END_VAR
TEST('TimeoutIncludesEntryAndSatisfiedConditions');
sm.ResetAll(); sm.ForceState(state := TcForge.E_SM_State.RUNNING); sm.SetCurrentStep(nStep := 3000); sm.SetTimerSeconds(seconds := 1.0);
step_TimeoutIncludesEntryAndSatisfiedConditions(sm := sm, nStep := 3000, nNextStep := 3002, nTimeout := 1, nRequired := 0);
AssertFalse(Condition := step_TimeoutIncludesEntryAndSatisfiedConditions.Entry OR step_TimeoutIncludesEntryAndSatisfiedConditions.Execute OR step_TimeoutIncludesEntryAndSatisfiedConditions.Exiting, Message := 'Timeout must suppress all lifecycle outputs even with no missing conditions');
AssertEquals_DINT(Expected := TcForge.E_SM_Fault.StepTimeout, Actual := sm.GetFaultCode(), Message := 'Timeout at the configured boundary');
TEST_FINISHED();
END_METHOD

METHOD StopTimeoutEscalatesToAbort
VAR

END_VAR
TEST('StopTimeoutEscalatesToAbort');
sm.ResetAll(); sm.ForceState(state := TcForge.E_SM_State.STOPPING); sm.SetCurrentStep(nStep := 2000); sm.ForceNextStep(nStep := 2000); sm.SetTimerSeconds(seconds := 2.0);
step_StopTimeoutEscalatesToAbort(sm := sm, nStep := 2000, nNextStep := 0, nTimeout := 1);
sm();
AssertEquals_DINT(Expected := TcForge.E_SM_State.ABORTING, Actual := sm.Status.State, Message := 'Failed Stop must escalate');
AssertEquals_DINT(Expected := 5000, Actual := sm.Status.Step.Current, Message := 'Abort entry step selected immediately');
AssertTrue(Condition := sm.IsFaulted(), Message := 'Escalation must preserve failure diagnostics');
TEST_FINISHED();
END_METHOD

METHOD StopUserFaultEscalatesToAbort
VAR

END_VAR
TEST('StopUserFaultEscalatesToAbort');
sm.ResetAll(); sm.ForceState(state := TcForge.E_SM_State.STOPPING); sm.SetCurrentStep(nStep := 2000); sm.ForceNextStep(nStep := 2000);
step_StopUserFaultEscalatesToAbort(sm := sm, nStep := 2000, nNextStep := 0, nTimeout := 0);
step_StopUserFaultEscalatesToAbort.RaiseFault(code := 101, reason := 'Stop feedback failed'); sm();
AssertEquals_DINT(Expected := TcForge.E_SM_State.ABORTING, Actual := sm.Status.State, Message := 'Custom shutdown fault must escalate independently of diagnostic code');
TEST_FINISHED();
END_METHOD

METHOD AbortTimeoutRequiresConfirmedShutdown
VAR
rsp : TcForge.E_RpcMethodResponse;
END_VAR
TEST('AbortTimeoutRequiresConfirmedShutdown');
sm.ResetAll(); sm.ForceState(state := TcForge.E_SM_State.ABORTING); sm.SetCurrentStep(nStep := 5000); sm.ForceNextStep(nStep := 5000); sm.SetTimerSeconds(seconds := 2.0);
step_AbortTimeoutRequiresConfirmedShutdown(sm := sm, nStep := 5000, nNextStep := 0, nTimeout := 1); sm();
AssertEquals_DINT(Expected := TcForge.E_SM_State.STOPPED, Actual := sm.Status.State, Message := 'Failed Abort must leave a defined terminal state');
AssertTrue(Condition := sm.Status.ShutdownFailed AND sm.IsFaulted(), Message := 'Terminal state must not masquerade as confirmed shutdown');
rsp := sm.Reset();
AssertEquals_DINT(Expected := TcForge.E_RpcMethodResponse.REJECTED_INTERLOCKED, Actual := rsp, Message := 'Reset requires application shutdown confirmation');
sm.inpShutdownConfirmed := TRUE; rsp := sm.Reset();
AssertEquals_DINT(Expected := TcForge.E_RpcMethodResponse.ACCEPTED, Actual := rsp, Message := 'Confirmed healthy terminal shutdown permits Reset');
AssertFalse(Condition := sm.Status.ShutdownFailed OR sm.IsFaulted(), Message := 'Reset clears the latched shutdown diagnostic');
TEST_FINISHED();
END_METHOD

METHOD CustomStepFaultCanRetry
VAR
rsp : TcForge.E_RpcMethodResponse;
END_VAR
TEST('CustomStepFaultCanRetry');
sm.ResetAll(); sm.ForceState(state := TcForge.E_SM_State.RUNNING); sm.SetCurrentStep(nStep := 3000); sm.ForceNextStep(nStep := 3000);
step_CustomStepFaultCanRetry(sm := sm, nStep := 3000, nNextStep := 3002, nTimeout := 0); step_CustomStepFaultCanRetry.RaiseFault(code := 101, reason := 'Application fault'); sm();
rsp := sm.Retry(); AssertEquals_DINT(Expected := TcForge.E_RpcMethodResponse.ACCEPTED, Actual := rsp, Message := 'Recorded custom step faults must support explicit retry');
sm(); sm(); AssertEquals_DINT(Expected := 3000, Actual := sm.Status.Step.Current, Message := 'Retry returns to failed even step');
TEST_FINISHED();
END_METHOD

METHOD MissingActiveStepFaults
VAR

END_VAR
TEST('MissingActiveStepFaults');
missing(); missing.Home(); missing(); missing();
AssertEquals_DINT(Expected := TcForge.E_SM_Fault.MissingStepImplementation, Actual := missing.GetFaultCode(), Message := 'Uncalled active step cannot silently stall');
AssertEquals_DINT(Expected := 1000, Actual := missing.Status.FailedStep, Message := 'Identify the missing implementation');
TEST_FINISHED();
END_METHOD

METHOD DuplicateActiveStepFaults
VAR

END_VAR
TEST('DuplicateActiveStepFaults');
duplicate(); duplicate.Home(); duplicate();
duplicateA(sm := duplicate, nStep := 1000, nNextStep := 0, nTimeout := 0);
duplicateB(sm := duplicate, nStep := 1000, nNextStep := 0, nTimeout := 0);
duplicate();
AssertEquals_DINT(Expected := TcForge.E_SM_Fault.DuplicateStepImplementation, Actual := duplicate.GetFaultCode(), Message := 'Two implementations of the active step must fault');
TEST_FINISHED();
END_METHOD

METHOD MissingDestinationImplementationFaults
VAR
i : INT;
END_VAR
TEST('MissingDestinationImplementationFaults');
missingTarget(); missingTarget.Home(); missingTarget();
FOR i := 1 TO 5 DO
    targetStep(sm := missingTarget, nStep := 1000, nNextStep := 1002, nTimeout := 0);
    missingTarget();
END_FOR;
AssertEquals_DINT(Expected := TcForge.E_SM_Fault.MissingStepImplementation, Actual := missingTarget.GetFaultCode(), Message := 'Valid but unimplemented destination must fault');
AssertEquals_DINT(Expected := 1002, Actual := missingTarget.Status.FailedStep, Message := 'Report destination without implementation');
TEST_FINISHED();
END_METHOD

METHOD MissingAbortImplementationFailsShutdown
VAR

END_VAR
TEST('MissingAbortImplementationFailsShutdown');
missingAbort(); missingAbort.Home(); missingAbort(); missingAbort.Abort(); missingAbort(); missingAbort();
AssertEquals_DINT(Expected := TcForge.E_SM_State.STOPPED, Actual := missingAbort.Status.State, Message := 'Missing Abort cannot leave a stuck state');
AssertTrue(Condition := missingAbort.Status.ShutdownFailed, Message := 'Missing Abort requires confirmed recovery');
TEST_FINISHED();
END_METHOD

METHOD StepZeroNeverExecutes
VAR

END_VAR
TEST('StepZeroNeverExecutes');
zero(); zeroStep(sm := zero, nStep := 0, nNextStep := 0, nTimeout := 0);
AssertFalse(Condition := zeroStep.Entry OR zeroStep.Execute OR zeroStep.Exiting, Message := 'Idle step zero is not executable work');
TEST_FINISHED();
END_METHOD

METHOD TimeoutAboveTimerRangeRejected
VAR

END_VAR
TEST('TimeoutAboveTimerRangeRejected');
sm.ResetAll(); sm.ForceState(state := TcForge.E_SM_State.RUNNING); sm.SetCurrentStep(nStep := 3000);
extraTimeout(sm := sm, nStep := 3000, nNextStep := 0, nTimeout := 356401);
AssertFalse(Condition := extraTimeout.Entry, Message := 'Unsupported timeout cannot silently wait forever');
AssertEquals_DINT(Expected := TcForge.E_SM_Fault.InvalidStepConfiguration, Actual := sm.GetFaultCode(), Message := 'Timeout above timer range is invalid');
TEST_FINISHED();
END_METHOD

METHOD ZeroFaultCodeStillInhibits
VAR

END_VAR
TEST('ZeroFaultCodeStillInhibits');
sm.ResetAll(); sm.ForceState(state := TcForge.E_SM_State.RUNNING); sm.SetCurrentStep(nStep := 3000);
extraZero(sm := sm, nStep := 3000, nNextStep := 0, nTimeout := 0); extraZero.RaiseFault(code := 0, reason := 'Invalid application code');
AssertTrue(Condition := sm.IsFaulted(), Message := 'Zero cannot hide a requested fault');
AssertFalse(Condition := extraZero.Entry OR extraZero.Execute OR extraZero.Exiting, Message := 'Fault immediately removes lifecycle outputs');
AssertEquals_DINT(Expected := TcForge.E_SM_Fault.StepUserFault, Actual := sm.GetFaultCode(), Message := 'Normalize invalid code');
TEST_FINISHED();
END_METHOD

METHOD NegativeFaultCodeStillInhibits
VAR

END_VAR
TEST('NegativeFaultCodeStillInhibits');
sm.ResetAll(); sm.ForceState(state := TcForge.E_SM_State.RUNNING); sm.SetCurrentStep(nStep := 3000);
extraNegative(sm := sm, nStep := 3000, nNextStep := 0, nTimeout := 0); extraNegative.RaiseFault(code := -1, reason := 'Invalid application code');
AssertTrue(Condition := sm.IsFaulted(), Message := 'Negative code cannot hide a requested fault');
AssertEquals_DINT(Expected := TcForge.E_SM_Fault.StepUserFault, Actual := sm.GetFaultCode(), Message := 'Normalize invalid code');
TEST_FINISHED();
END_METHOD

METHOD InvalidResetPreservesShutdownLatch
VAR
raw : DINT := 99;
requester : POINTER TO TcForge.E_Requester;
rsp : TcForge.E_RpcMethodResponse;
END_VAR
TEST('InvalidResetPreservesShutdownLatch');
sm.ResetAll(); sm.ForceState(state := TcForge.E_SM_State.ABORTING); sm.SetCurrentStep(nStep := 5000); sm.ForceNextStep(nStep := 5000);
extraReset(sm := sm, nStep := 5000, nNextStep := 0, nTimeout := 0); extraReset.RaiseFault(code := 101, reason := 'Abort failed'); sm();
sm.inpShutdownConfirmed := TRUE;
requester := ADR(raw); rsp := sm.Reset(eRequester := requester^);
AssertEquals_DINT(Expected := TcForge.E_RpcMethodResponse.REJECTED_INVALID_PARAMETER, Actual := rsp, Message := 'Invalid command identity rejected');
AssertTrue(Condition := sm.Status.ShutdownFailed, Message := 'Rejected reset preserves shutdown latch');
AssertEquals_DINT(Expected := 5000, Actual := sm.Status.FailedStep, Message := 'Rejected reset preserves failed step');
TEST_FINISHED();
END_METHOD

END_FUNCTION_BLOCK

// ---- Testing/Tests/FB_Foundation_Test.TcPOU
FUNCTION_BLOCK FB_Foundation_Test EXTENDS TcUnit.FB_TestSuite
VAR
    _done : BOOL;
    RecordedFaultBlocksStart_sm : FB_StateMachine_Probe;
    RetryRecoversOddStep_sm : FB_StateMachine_Probe;
    StopHandlesPausedAndHoming_sm : FB_StateMachine_Probe;
    AbortCannotBeOverwritten_sm : FB_StateMachine_Probe;
    StopCancelsQueuedHome_sm : FB_StateMachine_Probe;
    PendingHomeRechecksPermissive_sm : FB_StateMachine_Probe;
    MissingRequiredPermissiveInhibits_fb : TcForge.FB_Permissives;
    MissingRequiredInterlockLatches_fb : TcForge.FB_Interlock;
    DigitalQualityRecoveryNeedsCommand_fb : TcForge.FB_DigitalOutput;
    ForceSafeBypassesInvertAndDelay_fb : TcForge.FB_DigitalOutput;
    OperatorCannotClaimProgram_fb : TcForge.FB_DigitalOutput;
    AnalogLiveConfigFaultInhibits_fb : TcForge.FB_AnalogOutput;
    AnalogQualityRecoveryNeedsCommand_fb : TcForge.FB_AnalogOutput;
    ActuatorTripDropsOutputSameScan_fb : TcForge.FB_TwoPosActuator;
    ActuatorAbortDoesNotReenergizeHold_fb : TcForge.FB_TwoPosActuator;
    ExternalInputUsesPublicBoundary_fb : TcForge.FB_DigitalInput;
    ResetDoesNotStopRunningMachine_sm : FB_StateMachine_Probe;
    PublicSequenceLifecycle_sm : TcForge.FB_StateMachine;
    PublicSequenceLifecycle_homeStep : TcForge.FB_Step;
    PublicSequenceLifecycle_stopStep : TcForge.FB_Step;
    RateAlarmSeedsAndDetectsChange_fb : TcForge.FB_AlarmRateOfChange;
    StartupDoesNotRestoreWithoutOptIn_fb : FB_OutputRestart_Probe;
    StartupRestoreRequiresGoodQuality_fb : FB_OutputRestart_Probe;
    StartupRestoreRequiresGoodQuality_restored : FB_OutputRestart_Probe;
    SubmoduleFaultDoesNotPreventAbortCompletion_sm : FB_StateMachine_Probe;
    ActuatorAbortDominatesSameScan_fb : TcForge.FB_TwoPosActuator;
END_VAR

IF _done THEN RETURN; END_IF;
RecordedFaultBlocksStart();
RetryRecoversOddStep();
StopHandlesPausedAndHoming();
AbortCannotBeOverwritten();
StopCancelsQueuedHome();
PendingHomeRechecksPermissive();
MissingRequiredPermissiveInhibits();
MissingRequiredInterlockLatches();
DigitalQualityRecoveryNeedsCommand();
ForceSafeBypassesInvertAndDelay();
OperatorCannotClaimProgram();
AnalogLiveConfigFaultInhibits();
AnalogQualityRecoveryNeedsCommand();
ActuatorTripDropsOutputSameScan();
ActuatorAbortDoesNotReenergizeHold();
ExternalInputUsesPublicBoundary();
ResetDoesNotStopRunningMachine();
PublicSequenceLifecycle();
RateAlarmSeedsAndDetectsChange();
StartupDoesNotRestoreWithoutOptIn();
StartupRestoreRequiresGoodQuality();
SubmoduleFaultDoesNotPreventAbortCompletion();
ActuatorAbortDominatesSameScan();
_done := TRUE;

METHOD RecordedFaultBlocksStart
VAR
rsp : TcForge.E_RpcMethodResponse;
END_VAR
TEST('RecordedFaultBlocksStart');
RecordedFaultBlocksStart_sm.ResetAll(); RecordedFaultBlocksStart_sm.ForceState(state := TcForge.E_SM_State.READY); RecordedFaultBlocksStart_sm();
RecordedFaultBlocksStart_sm.inpSubmoduleFaulted := TRUE; RecordedFaultBlocksStart_sm();
rsp := RecordedFaultBlocksStart_sm.Start();
AssertEquals_DINT(Expected := TcForge.E_RpcMethodResponse.REJECTED_FAULTED, Actual := rsp, Message := 'Base fault must block Start even on an even step');
TEST_FINISHED();
END_METHOD

METHOD RetryRecoversOddStep
VAR
rsp : TcForge.E_RpcMethodResponse;
END_VAR
TEST('RetryRecoversOddStep');
RetryRecoversOddStep_sm.ResetAll(); RetryRecoversOddStep_sm.ForceState(state := TcForge.E_SM_State.RUNNING);
RetryRecoversOddStep_sm.SetCurrentStep(nStep := 3001); RetryRecoversOddStep_sm.ForceNextStep(nStep := 3001); RetryRecoversOddStep_sm();
rsp := RetryRecoversOddStep_sm.Retry();
AssertEquals_DINT(Expected := TcForge.E_RpcMethodResponse.ACCEPTED, Actual := rsp, Message := 'Retry must accept recovery step');
RetryRecoversOddStep_sm(); RetryRecoversOddStep_sm();
AssertEquals_DINT(Expected := 3000, Actual := RetryRecoversOddStep_sm.Status.Step.Current, Message := 'Retry re-enters previous even step');
AssertFalse(Condition := RetryRecoversOddStep_sm.IsFaulted(), Message := 'Recovered step fault must clear');
TEST_FINISHED();
END_METHOD

METHOD StopHandlesPausedAndHoming
VAR
i : INT;
rsp : TcForge.E_RpcMethodResponse;
END_VAR
TEST('StopHandlesPausedAndHoming');
FOR i := 0 TO 1 DO
StopHandlesPausedAndHoming_sm.ResetAll();
IF i = 0 THEN StopHandlesPausedAndHoming_sm.ForceState(state := TcForge.E_SM_State.PAUSED); ELSE StopHandlesPausedAndHoming_sm.ForceState(state := TcForge.E_SM_State.HOMING); END_IF;
rsp := StopHandlesPausedAndHoming_sm.Stop(); StopHandlesPausedAndHoming_sm();
AssertEquals_DINT(Expected := TcForge.E_RpcMethodResponse.ACCEPTED, Actual := rsp, Message := 'Stop is accepted');
AssertEquals_DINT(Expected := TcForge.E_SM_State.STOPPING, Actual := StopHandlesPausedAndHoming_sm.Status.State, Message := 'Accepted Stop starts stopping sequence');
END_FOR;
TEST_FINISHED();
END_METHOD

METHOD AbortCannotBeOverwritten
VAR
rsp : TcForge.E_RpcMethodResponse;
END_VAR
TEST('AbortCannotBeOverwritten');
AbortCannotBeOverwritten_sm.ResetAll(); AbortCannotBeOverwritten_sm.ForceState(state := TcForge.E_SM_State.RUNNING);
AbortCannotBeOverwritten_sm.Abort(); rsp := AbortCannotBeOverwritten_sm.Pause(); AbortCannotBeOverwritten_sm.Stop(); AbortCannotBeOverwritten_sm();
AssertEquals_DINT(Expected := TcForge.E_RpcMethodResponse.REJECTED_WRONG_STATE, Actual := rsp, Message := 'Pause cannot replace Abort');
AssertEquals_DINT(Expected := TcForge.E_SM_State.ABORTING, Actual := AbortCannotBeOverwritten_sm.Status.State, Message := 'Abort has priority');
TEST_FINISHED();
END_METHOD

METHOD StopCancelsQueuedHome
VAR
END_VAR
TEST('StopCancelsQueuedHome');
StopCancelsQueuedHome_sm.ResetAll(); StopCancelsQueuedHome_sm(); StopCancelsQueuedHome_sm.Home(); StopCancelsQueuedHome_sm.Stop(); StopCancelsQueuedHome_sm(); StopCancelsQueuedHome_sm();
AssertEquals_DINT(Expected := TcForge.E_SM_State.STOPPED, Actual := StopCancelsQueuedHome_sm.Status.State, Message := 'Queued home must not survive Stop');
TEST_FINISHED();
END_METHOD

METHOD PendingHomeRechecksPermissive
VAR
END_VAR
TEST('PendingHomeRechecksPermissive');
PendingHomeRechecksPermissive_sm.ResetAll(); PendingHomeRechecksPermissive_sm(); PendingHomeRechecksPermissive_sm.Home(); PendingHomeRechecksPermissive_sm.MapHomeCondition(bitIndex := 0, bGood := FALSE); PendingHomeRechecksPermissive_sm();
AssertEquals_DINT(Expected := TcForge.E_SM_State.STOPPED, Actual := PendingHomeRechecksPermissive_sm.Status.State, Message := 'Current bad permission cancels pending Home');
PendingHomeRechecksPermissive_sm.MapHomeCondition(bitIndex := 0, bGood := TRUE); PendingHomeRechecksPermissive_sm();
AssertEquals_DINT(Expected := TcForge.E_SM_State.STOPPED, Actual := PendingHomeRechecksPermissive_sm.Status.State, Message := 'Cancelled request must not restart later');
TEST_FINISHED();
END_METHOD

METHOD MissingRequiredPermissiveInhibits
VAR
i : INT;
END_VAR
TEST('MissingRequiredPermissiveInhibits');
MissingRequiredPermissiveInhibits_fb.cfg.nRequired := 1; MissingRequiredPermissiveInhibits_fb();
AssertFalse(Condition := MissingRequiredPermissiveInhibits_fb.sts.bOK, Message := 'Never-mapped required condition must inhibit');
MissingRequiredPermissiveInhibits_fb.MapInput(bitIndex := 0, inputValue := TRUE); MissingRequiredPermissiveInhibits_fb();
AssertTrue(Condition := MissingRequiredPermissiveInhibits_fb.sts.bOK, Message := 'Fresh required condition is good');
FOR i := 1 TO 12 DO MissingRequiredPermissiveInhibits_fb(); END_FOR;
AssertFalse(Condition := MissingRequiredPermissiveInhibits_fb.sts.bOK, Message := 'Stale required condition must inhibit');
AssertEquals_ULINT(Expected := 1, Actual := MissingRequiredPermissiveInhibits_fb.sts.nMissing, Message := 'Missing mask identifies condition');
TEST_FINISHED();
END_METHOD

METHOD MissingRequiredInterlockLatches
VAR
i : INT;
END_VAR
TEST('MissingRequiredInterlockLatches');
MissingRequiredInterlockLatches_fb.cfg.nRequired := 1; MissingRequiredInterlockLatches_fb.MapInput(bitIndex := 0, inputValue := TRUE); MissingRequiredInterlockLatches_fb();
FOR i := 1 TO 12 DO MissingRequiredInterlockLatches_fb(); END_FOR;
MissingRequiredInterlockLatches_fb.MapInput(bitIndex := 0, inputValue := TRUE); MissingRequiredInterlockLatches_fb();
AssertFalse(Condition := MissingRequiredInterlockLatches_fb.sts.bOK, Message := 'Recovered missing interlock requires Reset');
MissingRequiredInterlockLatches_fb.Reset(); MissingRequiredInterlockLatches_fb.MapInput(bitIndex := 0, inputValue := TRUE); MissingRequiredInterlockLatches_fb();
AssertTrue(Condition := MissingRequiredInterlockLatches_fb.sts.bOK, Message := 'Reset after fresh data releases missing latch');
TEST_FINISHED();
END_METHOD

METHOD DigitalQualityRecoveryNeedsCommand
VAR
END_VAR
TEST('DigitalQualityRecoveryNeedsCommand');
DigitalQualityRecoveryNeedsCommand_fb.SetOn(); DigitalQualityRecoveryNeedsCommand_fb(); AssertTrue(Condition := DigitalQualityRecoveryNeedsCommand_fb.sts.value, Message := 'Output starts on command');
DigitalQualityRecoveryNeedsCommand_fb(inpQuality := TcForge.E_IO_Quality.BAD);
AssertFalse(Condition := DigitalQualityRecoveryNeedsCommand_fb.sts.value, Message := 'Default bad-quality policy applies safe level');
DigitalQualityRecoveryNeedsCommand_fb(inpQuality := TcForge.E_IO_Quality.GOOD);
AssertFalse(Condition := DigitalQualityRecoveryNeedsCommand_fb.sts.value, Message := 'Quality recovery alone must not energize');
DigitalQualityRecoveryNeedsCommand_fb.SetOn(); DigitalQualityRecoveryNeedsCommand_fb(); AssertTrue(Condition := DigitalQualityRecoveryNeedsCommand_fb.sts.value, Message := 'Fresh command resumes output');
TEST_FINISHED();
END_METHOD

METHOD ForceSafeBypassesInvertAndDelay
VAR
rsp : TcForge.E_RpcMethodResponse;
END_VAR
TEST('ForceSafeBypassesInvertAndDelay');
ForceSafeBypassesInvertAndDelay_fb.cfg.invert := TRUE; ForceSafeBypassesInvertAndDelay_fb.cfg.debounceOff := T#10S;
ForceSafeBypassesInvertAndDelay_fb.SetOff(); ForceSafeBypassesInvertAndDelay_fb(); ForceSafeBypassesInvertAndDelay_fb.ForceSafe(); rsp := ForceSafeBypassesInvertAndDelay_fb.SetOn(); ForceSafeBypassesInvertAndDelay_fb();
AssertEquals_DINT(Expected := TcForge.E_RpcMethodResponse.REJECTED_INTERLOCKED, Actual := rsp, Message := 'ForceSafe wins within scan');
AssertFalse(Condition := ForceSafeBypassesInvertAndDelay_fb.sts.value, Message := 'ForceSafe writes electrical safe level without invert/delay');
TEST_FINISHED();
END_METHOD

METHOD OperatorCannotClaimProgram
VAR
rsp : TcForge.E_RpcMethodResponse;
END_VAR
TEST('OperatorCannotClaimProgram');
OperatorCannotClaimProgram_fb();
OperatorCannotClaimProgram_fb.LockSource(bLock := TRUE); rsp := OperatorCannotClaimProgram_fb.OperatorSetOn(requestId := 1);
AssertEquals_DINT(Expected := TcForge.E_RpcMethodResponse.QUEUED, Actual := rsp, Message := 'Admission is not execution');
OperatorCannotClaimProgram_fb();
rsp := OperatorCannotClaimProgram_fb.OperatorCommandResult(requestId := 1);
AssertEquals_DINT(Expected := TcForge.E_RpcMethodResponse.REJECTED_SOURCE_NOT_ALLOWED, Actual := rsp, Message := 'Operator wrapper always uses OPERATOR identity');
TEST_FINISHED();
END_METHOD

METHOD AnalogLiveConfigFaultInhibits
VAR
END_VAR
TEST('AnalogLiveConfigFaultInhibits');
AnalogLiveConfigFaultInhibits_fb.SetValue(rValue := 50.0); AnalogLiveConfigFaultInhibits_fb(); AnalogLiveConfigFaultInhibits_fb.cfg.euMax := AnalogLiveConfigFaultInhibits_fb.cfg.euMin; AnalogLiveConfigFaultInhibits_fb();
AssertTrue(Condition := AnalogLiveConfigFaultInhibits_fb.IsFaulted(), Message := 'Live invalid range must fault');
AssertTrue(Condition := AnalogLiveConfigFaultInhibits_fb.sts.outputInhibited, Message := 'Invalid config inhibits output same scan');
AssertTrue(Condition := AnalogLiveConfigFaultInhibits_fb.sts.rawReal = 0.0, Message := 'Fallback is raw safe value');
TEST_FINISHED();
END_METHOD

METHOD AnalogQualityRecoveryNeedsCommand
VAR
END_VAR
TEST('AnalogQualityRecoveryNeedsCommand');
AnalogQualityRecoveryNeedsCommand_fb.SetValue(rValue := 50.0); AnalogQualityRecoveryNeedsCommand_fb(); AnalogQualityRecoveryNeedsCommand_fb(inpQuality := TcForge.E_IO_Quality.UNKNOWN); AnalogQualityRecoveryNeedsCommand_fb(inpQuality := TcForge.E_IO_Quality.GOOD);
AssertTrue(Condition := AnalogQualityRecoveryNeedsCommand_fb.sts.outputInhibited, Message := 'Unknown quality disarms until fresh command');
AnalogQualityRecoveryNeedsCommand_fb.SetValue(rValue := 25.0); AnalogQualityRecoveryNeedsCommand_fb();
AssertFalse(Condition := AnalogQualityRecoveryNeedsCommand_fb.sts.outputInhibited, Message := 'Fresh command re-arms');
TEST_FINISHED();
END_METHOD

METHOD ActuatorTripDropsOutputSameScan
VAR
END_VAR
TEST('ActuatorTripDropsOutputSameScan');
ActuatorTripDropsOutputSameScan_fb(inAdvanced := FALSE, inRetracted := TRUE);
ActuatorTripDropsOutputSameScan_fb.Advance(); ActuatorTripDropsOutputSameScan_fb(); AssertTrue(Condition := ActuatorTripDropsOutputSameScan_fb.outAdvance, Message := 'Motion output energized');
ActuatorTripDropsOutputSameScan_fb(inAdvanced := TRUE, inRetracted := TRUE);
AssertTrue(Condition := ActuatorTripDropsOutputSameScan_fb.IsFaulted(), Message := 'Contradictory feedback faults');
AssertFalse(Condition := ActuatorTripDropsOutputSameScan_fb.outAdvance OR ActuatorTripDropsOutputSameScan_fb.outRetract, Message := 'Fault removes both outputs same scan');
TEST_FINISHED();
END_METHOD

METHOD ActuatorAbortDoesNotReenergizeHold
VAR
END_VAR
TEST('ActuatorAbortDoesNotReenergizeHold');
ActuatorAbortDoesNotReenergizeHold_fb.cfg.holdAtRetracted := TRUE; ActuatorAbortDoesNotReenergizeHold_fb(inRetracted := TRUE);
ActuatorAbortDoesNotReenergizeHold_fb.Abort(); ActuatorAbortDoesNotReenergizeHold_fb(); ActuatorAbortDoesNotReenergizeHold_fb();
AssertFalse(Condition := ActuatorAbortDoesNotReenergizeHold_fb.outRetract, Message := 'Abort must not automatically energize hold coil later');
TEST_FINISHED();
END_METHOD

METHOD ExternalInputUsesPublicBoundary
VAR
END_VAR
TEST('ExternalInputUsesPublicBoundary');
ExternalInputUsesPublicBoundary_fb(inSignal := TRUE);
AssertTrue(Condition := ExternalInputUsesPublicBoundary_fb.sts.value, Message := 'Digital external input path works without probe');
TEST_FINISHED();
END_METHOD

METHOD ResetDoesNotStopRunningMachine
VAR
rsp : TcForge.E_RpcMethodResponse;
END_VAR
TEST('ResetDoesNotStopRunningMachine');
ResetDoesNotStopRunningMachine_sm.ResetAll(); ResetDoesNotStopRunningMachine_sm.ForceState(state := TcForge.E_SM_State.RUNNING); rsp := ResetDoesNotStopRunningMachine_sm.Reset();
AssertEquals_DINT(Expected := TcForge.E_RpcMethodResponse.REJECTED_WRONG_STATE, Actual := rsp, Message := 'Reset requires stopped state');
TEST_FINISHED();
END_METHOD

METHOD PublicSequenceLifecycle
VAR
i : INT;
END_VAR
TEST('PublicSequenceLifecycle');
PublicSequenceLifecycle_sm(); PublicSequenceLifecycle_sm.Home(); PublicSequenceLifecycle_sm();
AssertEquals_DINT(Expected := 1000, Actual := PublicSequenceLifecycle_sm.Status.Step.Current, Message := 'Home enters first step');
FOR i := 1 TO 5 DO
    PublicSequenceLifecycle_homeStep(sm := PublicSequenceLifecycle_sm, nStep := 1000, nNextStep := 0, nTimeout := 0, sName := 'Home'); PublicSequenceLifecycle_sm();
END_FOR;
AssertEquals_DINT(Expected := TcForge.E_SM_State.READY, Actual := PublicSequenceLifecycle_sm.Status.State, Message := 'Home completion enters ready');
PublicSequenceLifecycle_sm.Start(); PublicSequenceLifecycle_sm(); PublicSequenceLifecycle_sm.Stop(); PublicSequenceLifecycle_sm();
FOR i := 1 TO 5 DO
    PublicSequenceLifecycle_stopStep(sm := PublicSequenceLifecycle_sm, nStep := 2000, nNextStep := 0, nTimeout := 0, sName := 'Stop'); PublicSequenceLifecycle_sm();
END_FOR;
AssertEquals_DINT(Expected := TcForge.E_SM_State.STOPPED, Actual := PublicSequenceLifecycle_sm.Status.State, Message := 'Stop sequence completes through public API');
PublicSequenceLifecycle_sm(); AssertEquals_DINT(Expected := TcForge.E_SM_State.STOPPED, Actual := PublicSequenceLifecycle_sm.Status.State, Message := 'No stale commands replay');
TEST_FINISHED();
END_METHOD

METHOD RateAlarmSeedsAndDetectsChange
VAR
END_VAR
TEST('RateAlarmSeedsAndDetectsChange');
RateAlarmSeedsAndDetectsChange_fb.cfg.common.bEnable := TRUE; RateAlarmSeedsAndDetectsChange_fb.cfg.fRateLimit := 1.0;
RateAlarmSeedsAndDetectsChange_fb(inpPv := 100.0); AssertTrue(Condition := RateAlarmSeedsAndDetectsChange_fb.outRateOfChange = 0.0, Message := 'First scan seeds rate');
RateAlarmSeedsAndDetectsChange_fb(inpPv := 200.0); AssertTrue(Condition := RateAlarmSeedsAndDetectsChange_fb.sts.active, Message := 'Fast change trips rate alarm');
RateAlarmSeedsAndDetectsChange_fb.cfg.common.bEnable := FALSE; RateAlarmSeedsAndDetectsChange_fb(); RateAlarmSeedsAndDetectsChange_fb.cfg.common.bEnable := TRUE; RateAlarmSeedsAndDetectsChange_fb(inpPv := 999.0);
AssertTrue(Condition := RateAlarmSeedsAndDetectsChange_fb.outRateOfChange = 0.0, Message := 'Re-enable reseeds rate');
TEST_FINISHED();
END_METHOD

METHOD StartupDoesNotRestoreWithoutOptIn
VAR
END_VAR
TEST('StartupDoesNotRestoreWithoutOptIn');
StartupDoesNotRestoreWithoutOptIn_fb.SeedSavedCommand(value := TRUE); StartupDoesNotRestoreWithoutOptIn_fb();
AssertFalse(Condition := StartupDoesNotRestoreWithoutOptIn_fb.sts.value, Message := 'Saved command does not implicitly restore output');
TEST_FINISHED();
END_METHOD

METHOD StartupRestoreRequiresGoodQuality
VAR
END_VAR
TEST('StartupRestoreRequiresGoodQuality');
StartupRestoreRequiresGoodQuality_fb.SeedSavedCommand(value := TRUE); StartupRestoreRequiresGoodQuality_fb.cfg.restoreCommandOnRestart := TRUE; StartupRestoreRequiresGoodQuality_fb(inpQuality := TcForge.E_IO_Quality.BAD); StartupRestoreRequiresGoodQuality_fb(inpQuality := TcForge.E_IO_Quality.GOOD);
AssertFalse(Condition := StartupRestoreRequiresGoodQuality_fb.sts.value, Message := 'Bad startup quality cancels restoration');
StartupRestoreRequiresGoodQuality_restored.SeedSavedCommand(value := TRUE); StartupRestoreRequiresGoodQuality_restored.cfg.restoreCommandOnRestart := TRUE; StartupRestoreRequiresGoodQuality_restored();
AssertTrue(Condition := StartupRestoreRequiresGoodQuality_restored.sts.value, Message := 'Explicit opt-in restores with good startup quality');
TEST_FINISHED();
END_METHOD

METHOD SubmoduleFaultDoesNotPreventAbortCompletion
VAR
END_VAR
TEST('SubmoduleFaultDoesNotPreventAbortCompletion');
SubmoduleFaultDoesNotPreventAbortCompletion_sm.ResetAll(); SubmoduleFaultDoesNotPreventAbortCompletion_sm.ForceState(state := TcForge.E_SM_State.RUNNING); SubmoduleFaultDoesNotPreventAbortCompletion_sm.inpSubmoduleFaulted := TRUE; SubmoduleFaultDoesNotPreventAbortCompletion_sm();
SubmoduleFaultDoesNotPreventAbortCompletion_sm.ForceNextStep(nStep := 0); SubmoduleFaultDoesNotPreventAbortCompletion_sm();
AssertEquals_DINT(Expected := TcForge.E_SM_State.STOPPED, Actual := SubmoduleFaultDoesNotPreventAbortCompletion_sm.Status.State, Message := 'Persistent submodule fault must allow abort completion');
AssertTrue(Condition := SubmoduleFaultDoesNotPreventAbortCompletion_sm.IsFaulted(), Message := 'Completion does not erase submodule fault');
TEST_FINISHED();
END_METHOD

METHOD ActuatorAbortDominatesSameScan
VAR
    rsp : TcForge.E_RpcMethodResponse;
END_VAR
TEST('ActuatorAbortDominatesSameScan');
ActuatorAbortDominatesSameScan_fb(inRetracted := TRUE); ActuatorAbortDominatesSameScan_fb.Advance(); ActuatorAbortDominatesSameScan_fb(); ActuatorAbortDominatesSameScan_fb.Abort(); rsp := ActuatorAbortDominatesSameScan_fb.Advance(); ActuatorAbortDominatesSameScan_fb();
AssertEquals_DINT(Expected := TcForge.E_RpcMethodResponse.REJECTED_INTERLOCKED, Actual := rsp, Message := 'Abort cannot be replaced by motion in the same scan');
AssertFalse(Condition := ActuatorAbortDominatesSameScan_fb.outAdvance OR ActuatorAbortDominatesSameScan_fb.outRetract, Message := 'Abort leaves both coils off');
TEST_FINISHED();
END_METHOD

END_FUNCTION_BLOCK

// ---- Testing/Tests/FB_CyclicFoundation_Test.TcPOU
FUNCTION_BLOCK FB_CyclicFoundation_Test EXTENDS TcUnit.FB_TestSuite
VAR
    _pulse : TcForge.FB_DigitalOutput;
    _pulseClock : TON;
    _pulsePhase : UINT;
    _pulseDone : BOOL;
    _output : TcForge.FB_DigitalOutput;
    _actuator : TcForge.FB_TwoPosActuator;
    _timer : TON;
    _phase : UINT;
    _done : BOOL;
END_VAR

PulseLifecycle();
IF _done THEN RETURN; END_IF;
TEST('CyclicWatchdogAndMotionTimeout');
CASE _phase OF
0:
    _output.cfg.qualityFaultAfter := T#50MS;
    _output.SetOn(); _output();
    _actuator.cfg.advTimeoutS := 1;
    _actuator(inRetracted := TRUE);
    _actuator.Advance();
    _phase := 1;
1:
    _timer(IN := TRUE, PT := T#1500MS);
    _output(inpQuality := TcForge.E_IO_Quality.BAD);
    _actuator(inRetracted := FALSE, inAdvanced := FALSE);
    IF _timer.Q THEN
        AssertTrue(Condition := _output.IsFaulted(), Message := 'Real multi-scan watchdog expires');
        AssertFalse(Condition := _output.sts.value, Message := 'Faulted output stays safe');
        AssertEquals_DINT(Expected := TcForge.E_TwoPosActuator_Fault.AdvanceTimeout, Actual := _actuator.GetFaultCode(), Message := 'Travel timeout expires across scans');
        AssertFalse(Condition := _actuator.outAdvance OR _actuator.outRetract, Message := 'Timed-out actuator has no outputs');
        _output.Reset(); _output(inpQuality := TcForge.E_IO_Quality.GOOD);
        AssertFalse(Condition := _output.sts.value, Message := 'Reset does not restore saved command');
        _done := TRUE;
        TEST_FINISHED();
    END_IF;
END_CASE;

METHOD PulseLifecycle
IF _pulseDone THEN RETURN; END_IF;
TEST('CyclicDebounceAndSinglePulse');
CASE _pulsePhase OF
0:
    _pulse.cfg.mode := TcForge.E_DigitalOutput_Mode.SinglePulse;
    _pulse.cfg.debounceOn := T#50MS;
    _pulse.cfg.pulseOn := T#100MS;
    _pulse.SetOn(); _pulse();
    AssertFalse(Condition := _pulse.outSignal, Message := 'Debounce prevents an immediate pulse');
    _pulseClock(IN := TRUE, PT := T#2S);
    _pulsePhase := 1;
1:
    _pulseClock(IN := TRUE, PT := T#2S); _pulse();
    IF _pulse.outSignal THEN
        _pulseClock(IN := FALSE);
        _pulsePhase := 2;
    ELSIF _pulseClock.Q THEN
        AssertTrue(Condition := FALSE, Message := 'Pulse did not start within two seconds');
        _pulseDone := TRUE; TEST_FINISHED();
    END_IF;
2:
    _pulseClock(IN := TRUE, PT := T#300MS); _pulse();
    IF _pulseClock.Q THEN
        AssertFalse(Condition := _pulse.outSignal, Message := 'Single pulse ends and held command cannot retrigger it');
        _pulseDone := TRUE; TEST_FINISHED();
    END_IF;
END_CASE;
END_METHOD

END_FUNCTION_BLOCK

// ---- Testing/Tests/FB_F_ValidateRequester_Test.TcPOU
FUNCTION_BLOCK FB_F_ValidateRequester_Test EXTENDS TcUnit.FB_TestSuite
VAR
END_VAR

AcceptsNormally();
AcceptsProgramWhenLocked();
RejectsOperatorWhenLocked();
RejectsWhenFaulted();

METHOD AcceptsNormally
VAR
    nExpected : DINT := TcForge.E_RpcMethodResponse.ACCEPTED;
    nActual   : DINT;
END_VAR
TEST('AcceptsNormally');

nActual := TcForge.F_ValidateRequester(
    eRequester    := TcForge.E_Requester.OPERATOR,
    bSourceLocked := FALSE,
    bFaulted      := FALSE);

AssertEquals_DINT(
    Expected := nExpected,
    Actual   := nActual,
    Message  := 'Should accept when there are no restrictions');

TEST_FINISHED();
END_METHOD

METHOD AcceptsProgramWhenLocked
VAR
    nExpected : DINT := TcForge.E_RpcMethodResponse.ACCEPTED;
    nActual   : DINT;
END_VAR
TEST('AcceptsProgramWhenLocked');

nActual := TcForge.F_ValidateRequester(
    eRequester    := TcForge.E_Requester.PROG,
    bSourceLocked := TRUE,
    bFaulted      := FALSE);

AssertEquals_DINT(
    Expected := nExpected,
    Actual   := nActual,
    Message  := 'PROG requester should be accepted even when source is locked');

TEST_FINISHED();
END_METHOD

METHOD RejectsOperatorWhenLocked
VAR
    nExpected : DINT := TcForge.E_RpcMethodResponse.REJECTED_SOURCE_NOT_ALLOWED;
    nActual   : DINT;
END_VAR
TEST('RejectsOperatorWhenLocked');

nActual := TcForge.F_ValidateRequester(
    eRequester    := TcForge.E_Requester.OPERATOR,
    bSourceLocked := TRUE,
    bFaulted      := FALSE);

AssertEquals_DINT(
    Expected := nExpected,
    Actual   := nActual,
    Message  := 'OPERATOR must be rejected when source is locked');

TEST_FINISHED();
END_METHOD

METHOD RejectsWhenFaulted
VAR
    nExpected : DINT := TcForge.E_RpcMethodResponse.REJECTED_FAULTED;
    nActual   : DINT;
END_VAR
TEST('RejectsWhenFaulted');

nActual := TcForge.F_ValidateRequester(
    eRequester    := TcForge.E_Requester.OPERATOR,
    bSourceLocked := FALSE,
    bFaulted      := TRUE);

AssertEquals_DINT(
    Expected := nExpected,
    Actual   := nActual,
    Message  := 'Should reject when faulted');

TEST_FINISHED();
END_METHOD

END_FUNCTION_BLOCK

// ---- Testing/Tests/FB_BitMatrix64_Test.TcPOU
// Unit tests for FB_BitMatrix64 — the shared 64-bit condition-matrix core
// consumed by FB_Permissives (non-latching) and FB_Interlock (latching).
// Covers the behaviours both composers rely on: live bit semantics, active-
// mask tracking, mapping timeout, "just unmapped while bad" events, first-
// failure ordering, bypass accept/reject rules, and clear operations.
//
// Each test owns a fresh FB_BitMatrix64 instance via METHOD-local VARs so
// cycle counters and internal state do not leak between tests.
FUNCTION_BLOCK FB_BitMatrix64_Test EXTENDS TcUnit.FB_TestSuite

InitialStateAllGood();
MapInputMarksActiveAndValue();
MapInputBadValueClearsLiveBit();
MapInputOutOfRangeIsNoOp();
MappingTimeoutUnmapsAndRestoresGood();
JustUnmappedBadFiresWhenBadAtUnmap();
JustUnmappedBadSilentWhenGoodAtUnmap();
FirstFailureRecordsFirstBadBit();
SetBypassAcceptsWhenBypassable();
SetBypassRejectsWhenNotBypassable();
SetBypassClearAlwaysAllowed();
SetBypassInvalidBitIndex();
ClearBypassClearsAll();
ClearFirstFailureResets();

METHOD InitialStateAllGood
VAR
    fb : TcForge.FB_BitMatrix64;
END_VAR
TEST('InitialStateAllGood');

// Before any body call, default initialisers should mark every bit good
// and no bit active / bypassed / tripped.
AssertEquals_ULINT(
    Expected := 16#FFFFFFFFFFFFFFFF,
    Actual   := fb.nLiveBits,
    Message  := 'Fresh instance: nLiveBits should be all-good');
AssertEquals_ULINT(
    Expected := 0,
    Actual   := fb.nActiveMask,
    Message  := 'Fresh instance: nActiveMask should be empty');
AssertEquals_ULINT(
    Expected := 0,
    Actual   := fb.nBypassMask,
    Message  := 'Fresh instance: nBypassMask should be empty');
AssertEquals_UDINT(
    Expected := 999,
    Actual   := fb.nFirstFailureBitIndex,
    Message  := 'Fresh instance: nFirstFailureBitIndex should be sentinel 999');
AssertEquals_ULINT(
    Expected := 0,
    Actual   := fb.nJustUnmappedBad,
    Message  := 'Fresh instance: nJustUnmappedBad should be empty');

TEST_FINISHED();
END_METHOD

METHOD MapInputMarksActiveAndValue
VAR
    fb      : TcForge.FB_BitMatrix64;
    bitMask : ULINT;
END_VAR
TEST('MapInputMarksActiveAndValue');

bitMask := SHL(ULINT#1, 5);

fb.MapInput(bitIndex := 5, inputValue := TRUE);
fb();

AssertTrue(
    Condition := (fb.nActiveMask AND bitMask) <> 0,
    Message   := 'Bit 5 should be in nActiveMask after MapInput(5, TRUE)');
AssertTrue(
    Condition := (fb.nLiveBits AND bitMask) <> 0,
    Message   := 'Bit 5 should be good (1) in nLiveBits after MapInput(5, TRUE)');

TEST_FINISHED();
END_METHOD

METHOD MapInputBadValueClearsLiveBit
VAR
    fb      : TcForge.FB_BitMatrix64;
    bitMask : ULINT;
END_VAR
TEST('MapInputBadValueClearsLiveBit');

bitMask := SHL(ULINT#1, 5);

fb.MapInput(bitIndex := 5, inputValue := FALSE);
fb();

AssertTrue(
    Condition := (fb.nActiveMask AND bitMask) <> 0,
    Message   := 'Bit 5 should still be active even when value is FALSE');
AssertTrue(
    Condition := (fb.nLiveBits AND bitMask) = 0,
    Message   := 'Bit 5 should be bad (0) in nLiveBits after MapInput(5, FALSE)');

TEST_FINISHED();
END_METHOD

METHOD MapInputOutOfRangeIsNoOp
VAR
    fb : TcForge.FB_BitMatrix64;
END_VAR
TEST('MapInputOutOfRangeIsNoOp');

// Bit 64 is outside the 0..63 range; MapInput must silently reject it.
fb.MapInput(bitIndex := 64, inputValue := FALSE);
fb();

AssertEquals_ULINT(
    Expected := 0,
    Actual   := fb.nActiveMask,
    Message  := 'MapInput with bitIndex > 63 must not touch nActiveMask');
AssertEquals_ULINT(
    Expected := 16#FFFFFFFFFFFFFFFF,
    Actual   := fb.nLiveBits,
    Message  := 'MapInput with bitIndex > 63 must not touch nLiveBits');

TEST_FINISHED();
END_METHOD

METHOD MappingTimeoutUnmapsAndRestoresGood
VAR
    fb      : TcForge.FB_BitMatrix64;
    bitMask : ULINT;
    i       : UDINT;
END_VAR
TEST('MappingTimeoutUnmapsAndRestoresGood');

bitMask := SHL(ULINT#1, 5);

// Map bit 5 once as bad, then stop feeding. After MAPPING_TIMEOUT (=10)
// unreferenced cycles the bit must be unmapped and snap back to good.
fb.MapInput(bitIndex := 5, inputValue := FALSE);
fb();  // cycle 1 — freshly mapped

FOR i := 1 TO 12 DO  // run past the 10-cycle timeout
    fb();
END_FOR;

AssertTrue(
    Condition := (fb.nActiveMask AND bitMask) = 0,
    Message   := 'Bit 5 should be unmapped after MAPPING_TIMEOUT cycles without refresh');
AssertTrue(
    Condition := (fb.nLiveBits AND bitMask) <> 0,
    Message   := 'Bit 5 should snap back to good once unmapped');

TEST_FINISHED();
END_METHOD

METHOD JustUnmappedBadFiresWhenBadAtUnmap
VAR
    fb        : TcForge.FB_BitMatrix64;
    bitMask   : ULINT;
    i         : UDINT;
    sawEvent  : BOOL;
END_VAR
TEST('JustUnmappedBadFiresWhenBadAtUnmap');

bitMask := SHL(ULINT#1, 5);

// Map bit 5 as BAD, then stop feeding. Somewhere in the next cycles the
// cleanup loop will unmap it; that tick must publish the event via
// nJustUnmappedBad so latching callers (FB_Interlock) can remember it.
fb.MapInput(bitIndex := 5, inputValue := FALSE);
fb();

sawEvent := FALSE;
FOR i := 1 TO 15 DO
    fb();
    IF (fb.nJustUnmappedBad AND bitMask) <> 0 THEN
        sawEvent := TRUE;
    END_IF;
END_FOR;

AssertTrue(
    Condition := sawEvent,
    Message   := 'nJustUnmappedBad should fire for bit 5 during the timeout-unmap cycle');

// Event must be edge-style: once the unmap cycle passes, subsequent cycles
// reset the output.
AssertEquals_ULINT(
    Expected := 0,
    Actual   := fb.nJustUnmappedBad,
    Message  := 'nJustUnmappedBad should clear on cycles after the unmap event');

TEST_FINISHED();
END_METHOD

METHOD JustUnmappedBadSilentWhenGoodAtUnmap
VAR
    fb       : TcForge.FB_BitMatrix64;
    bitMask  : ULINT;
    i        : UDINT;
    sawEvent : BOOL;
END_VAR
TEST('JustUnmappedBadSilentWhenGoodAtUnmap');

bitMask := SHL(ULINT#1, 5);

// Map bit 5 as GOOD then stop feeding. The timeout unmap still happens,
// but there is no "bad at unmap" memory to expose — event must stay clear.
fb.MapInput(bitIndex := 5, inputValue := TRUE);
fb();

sawEvent := FALSE;
FOR i := 1 TO 15 DO
    fb();
    IF (fb.nJustUnmappedBad AND bitMask) <> 0 THEN
        sawEvent := TRUE;
    END_IF;
END_FOR;

AssertFalse(
    Condition := sawEvent,
    Message   := 'nJustUnmappedBad must NOT fire when the bit was good at unmap');

TEST_FINISHED();
END_METHOD

METHOD FirstFailureRecordsFirstBadBit
VAR
    fb : TcForge.FB_BitMatrix64;
END_VAR
TEST('FirstFailureRecordsFirstBadBit');

// Cycle 1: bits 3 and 7 both mapped good; baseline is all good.
fb.MapInput(bitIndex := 3, inputValue := TRUE);
fb.MapInput(bitIndex := 7, inputValue := TRUE);
fb();

// Cycle 2: both drop to bad in the same scan. The body scans bits 0..63 in
// order, so the lower-index bit (3) wins the first-failure slot.
fb.MapInput(bitIndex := 3, inputValue := FALSE);
fb.MapInput(bitIndex := 7, inputValue := FALSE);
fb();

AssertEquals_UDINT(
    Expected := 3,
    Actual   := fb.nFirstFailureBitIndex,
    Message  := 'First-failure index should be the lowest-numbered bit that went bad');

TEST_FINISHED();
END_METHOD

METHOD SetBypassAcceptsWhenBypassable
VAR
    fb       : TcForge.FB_BitMatrix64;
    bitMask  : ULINT;
    response : TcForge.E_RpcMethodResponse;
END_VAR
TEST('SetBypassAcceptsWhenBypassable');

bitMask := SHL(ULINT#1, 3);

response := fb.SetBypass(
    bitIndex        := 3,
    bEnable         := TRUE,
    nBypassableMask := bitMask);

AssertEquals_DINT(
    Expected := TcForge.E_RpcMethodResponse.ACCEPTED,
    Actual   := response,
    Message  := 'SetBypass should accept when the bit is configured as bypassable');
AssertTrue(
    Condition := (fb.nBypassMask AND bitMask) <> 0,
    Message   := 'nBypassMask should reflect the accepted bypass');

TEST_FINISHED();
END_METHOD

METHOD SetBypassRejectsWhenNotBypassable
VAR
    fb       : TcForge.FB_BitMatrix64;
    response : TcForge.E_RpcMethodResponse;
END_VAR
TEST('SetBypassRejectsWhenNotBypassable');

// Caller supplies an empty bypassable mask, so any enable attempt must be
// rejected regardless of which bit is targeted.
response := fb.SetBypass(
    bitIndex        := 3,
    bEnable         := TRUE,
    nBypassableMask := 0);

AssertEquals_DINT(
    Expected := TcForge.E_RpcMethodResponse.REJECTED_BYPASS_NOT_ALLOWED,
    Actual   := response,
    Message  := 'SetBypass must reject enable when the bit is not configured as bypassable');
AssertEquals_ULINT(
    Expected := 0,
    Actual   := fb.nBypassMask,
    Message  := 'nBypassMask must stay empty after a rejected SetBypass');

TEST_FINISHED();
END_METHOD

METHOD SetBypassClearAlwaysAllowed
VAR
    fb       : TcForge.FB_BitMatrix64;
    response : TcForge.E_RpcMethodResponse;
END_VAR
TEST('SetBypassClearAlwaysAllowed');

// Clearing a bypass is always safe: even if the bit is not configured as
// bypassable, removing a bypass cannot violate any safety invariant.
response := fb.SetBypass(
    bitIndex        := 3,
    bEnable         := FALSE,
    nBypassableMask := 0);

AssertEquals_DINT(
    Expected := TcForge.E_RpcMethodResponse.ACCEPTED,
    Actual   := response,
    Message  := 'Clearing a bypass must always be accepted');

TEST_FINISHED();
END_METHOD

METHOD SetBypassInvalidBitIndex
VAR
    fb       : TcForge.FB_BitMatrix64;
    response : TcForge.E_RpcMethodResponse;
END_VAR
TEST('SetBypassInvalidBitIndex');

response := fb.SetBypass(
    bitIndex        := 64,
    bEnable         := TRUE,
    nBypassableMask := 16#FFFFFFFFFFFFFFFF);

AssertEquals_DINT(
    Expected := TcForge.E_RpcMethodResponse.REJECTED_INVALID_PARAMETER,
    Actual   := response,
    Message  := 'SetBypass must reject bitIndex > 63 with REJECTED_INVALID_PARAMETER');

TEST_FINISHED();
END_METHOD

METHOD ClearBypassClearsAll
VAR
    fb : TcForge.FB_BitMatrix64;
END_VAR
TEST('ClearBypassClearsAll');

// Bypass two separate bits, then clear them in one call.
fb.SetBypass(bitIndex := 2, bEnable := TRUE, nBypassableMask := 16#FFFFFFFFFFFFFFFF);
fb.SetBypass(bitIndex := 9, bEnable := TRUE, nBypassableMask := 16#FFFFFFFFFFFFFFFF);
fb.ClearBypass();

AssertEquals_ULINT(
    Expected := 0,
    Actual   := fb.nBypassMask,
    Message  := 'ClearBypass must wipe nBypassMask in a single call');

TEST_FINISHED();
END_METHOD

METHOD ClearFirstFailureResets
VAR
    fb : TcForge.FB_BitMatrix64;
END_VAR
TEST('ClearFirstFailureResets');

// Produce a real first-failure sequence, then clear it.
fb.MapInput(bitIndex := 3, inputValue := TRUE);
fb();
fb.MapInput(bitIndex := 3, inputValue := FALSE);
fb();

AssertEquals_UDINT(
    Expected := 3,
    Actual   := fb.nFirstFailureBitIndex,
    Message  := 'Precondition: failure sequence should record bit 3');

fb.ClearFirstFailure();

AssertEquals_UDINT(
    Expected := 999,
    Actual   := fb.nFirstFailureBitIndex,
    Message  := 'ClearFirstFailure must restore the sentinel 999');

TEST_FINISHED();
END_METHOD

END_FUNCTION_BLOCK

// ---- Testing/Tests/FB_Permissives_Test.TcPOU
// Integration tests for FB_Permissives on top of FB_BitMatrix64.
// FB_BitMatrix64_Test already covers the shared matrix mechanics, so this
// suite focuses on permissive-specific behaviour:
//   - non-latching rollup: sts.bOK tracks live inputs in both directions
//   - bypass forces the bit good in the rollup
//   - Reset() clears bypass (the only thing Reset needs to do here — the
//     permissive has no latched state to snap)
//   - cfg.nBypassable gating propagates through SetBypass
//   - first-failure and faceplate surfaces reflect core state
FUNCTION_BLOCK FB_Permissives_Test EXTENDS TcUnit.FB_TestSuite

InitialStateOk();
BadMappedBitFailsOK();
RecoveryFlipsOKTrueAgain();
BypassForcesGoodInRollup();
ResetClearsBypass();
SetBypassRejectsWhenNotBypassable();
FirstFailureIndexPropagates();
FaceplateReflectsLiveState();

METHOD InitialStateOk
VAR
    fb : TcForge.FB_Permissives;
END_VAR
TEST('InitialStateOk');

fb();  // no MapInput calls — unmapped bits default good

AssertTrue(
    Condition := fb.sts.bOK,
    Message   := 'Fresh permissives with no mappings should report bOK = TRUE');
AssertEquals_ULINT(
    Expected := 16#FFFFFFFFFFFFFFFF,
    Actual   := fb.sts.nPermissives,
    Message  := 'Fresh permissives rollup should be all-good');
AssertEquals_UDINT(
    Expected := 999,
    Actual   := fb.sts.nFirstFailureBitIndex,
    Message  := 'Fresh permissives should expose the sentinel first-failure index');

TEST_FINISHED();
END_METHOD

METHOD BadMappedBitFailsOK
VAR
    fb      : TcForge.FB_Permissives;
    bitMask : ULINT;
END_VAR
TEST('BadMappedBitFailsOK');

bitMask := SHL(ULINT#1, 5);

fb.MapInput(bitIndex := 5, inputValue := FALSE);
fb();

AssertFalse(
    Condition := fb.sts.bOK,
    Message   := 'bOK must be FALSE when any mapped bit is bad');
AssertTrue(
    Condition := (fb.sts.nPermissives AND bitMask) = 0,
    Message   := 'Bit 5 should show as bad in the rollup');

TEST_FINISHED();
END_METHOD

METHOD RecoveryFlipsOKTrueAgain
VAR
    fb : TcForge.FB_Permissives;
END_VAR
TEST('RecoveryFlipsOKTrueAgain');

// This is the defining permissive behaviour: when the condition recovers,
// bOK returns to TRUE on the *same* cycle, with no Reset() required.
fb.MapInput(bitIndex := 5, inputValue := FALSE);
fb();

AssertFalse(
    Condition := fb.sts.bOK,
    Message   := 'Precondition: bOK should be FALSE while bit 5 is bad');

fb.MapInput(bitIndex := 5, inputValue := TRUE);
fb();

AssertTrue(
    Condition := fb.sts.bOK,
    Message   := 'Permissive is non-latching: bOK must flip back to TRUE the cycle the input recovers');

TEST_FINISHED();
END_METHOD

METHOD BypassForcesGoodInRollup
VAR
    fb       : TcForge.FB_Permissives;
    bitMask  : ULINT;
    response : TcForge.E_RpcMethodResponse;
END_VAR
TEST('BypassForcesGoodInRollup');

bitMask := SHL(ULINT#1, 5);
fb.cfg.nBypassable := bitMask;

fb.MapInput(bitIndex := 5, inputValue := FALSE);
response := fb.SetBypass(bitIndex := 5, bEnable := TRUE);
fb();

AssertEquals_DINT(
    Expected := TcForge.E_RpcMethodResponse.ACCEPTED,
    Actual   := response,
    Message  := 'SetBypass should accept when the bit is flagged bypassable in cfg');
AssertTrue(
    Condition := fb.sts.bOK,
    Message   := 'A bypassed bit must be forced good in the rollup');
AssertTrue(
    Condition := (fb.sts.nBypassMask AND bitMask) <> 0,
    Message   := 'sts.nBypassMask should surface the active bypass');

TEST_FINISHED();
END_METHOD

METHOD ResetClearsBypass
VAR
    fb      : TcForge.FB_Permissives;
    bitMask : ULINT;
END_VAR
TEST('ResetClearsBypass');

bitMask := SHL(ULINT#1, 3);
fb.cfg.nBypassable := bitMask;

fb.SetBypass(bitIndex := 3, bEnable := TRUE);
fb();

AssertTrue(
    Condition := (fb.sts.nBypassMask AND bitMask) <> 0,
    Message   := 'Precondition: bit 3 bypass should be active before Reset()');

fb.Reset();
fb();

AssertEquals_ULINT(
    Expected := 0,
    Actual   := fb.sts.nBypassMask,
    Message  := 'Reset() on a permissive must clear every bypass bit');

TEST_FINISHED();
END_METHOD

METHOD SetBypassRejectsWhenNotBypassable
VAR
    fb       : TcForge.FB_Permissives;
    response : TcForge.E_RpcMethodResponse;
END_VAR
TEST('SetBypassRejectsWhenNotBypassable');

fb.cfg.nBypassable := 0;

response := fb.SetBypass(bitIndex := 5, bEnable := TRUE);
fb();

AssertEquals_DINT(
    Expected := TcForge.E_RpcMethodResponse.REJECTED_BYPASS_NOT_ALLOWED,
    Actual   := response,
    Message  := 'SetBypass must honour cfg.nBypassable and reject non-allowed bits');
AssertEquals_ULINT(
    Expected := 0,
    Actual   := fb.sts.nBypassMask,
    Message  := 'A rejected bypass must leave nBypassMask untouched');

TEST_FINISHED();
END_METHOD

METHOD FirstFailureIndexPropagates
VAR
    fb : TcForge.FB_Permissives;
END_VAR
TEST('FirstFailureIndexPropagates');

fb.MapInput(bitIndex := 7, inputValue := TRUE);
fb();

fb.MapInput(bitIndex := 7, inputValue := FALSE);
fb();

AssertEquals_UDINT(
    Expected := 7,
    Actual   := fb.sts.nFirstFailureBitIndex,
    Message  := 'sts.nFirstFailureBitIndex should surface the core first-failure index');

TEST_FINISHED();
END_METHOD

METHOD FaceplateReflectsLiveState
VAR
    fb : TcForge.FB_Permissives;
END_VAR
TEST('FaceplateReflectsLiveState');

fb.cfg.nBypassable   := SHL(ULINT#1, 4);
fb.cfg.aNames[4]     := 'TestPerm';

fb.MapInput(bitIndex := 4, inputValue := FALSE);
fb();

AssertEquals_STRING(
    Expected := 'TestPerm',
    Actual   := fb.sts.aFaceplates[4].name,
    Message  := 'Faceplate should mirror cfg.aNames[i]');
AssertFalse(
    Condition := fb.sts.aFaceplates[4].ok,
    Message   := 'Faceplate ok should mirror the rollup for that bit');
AssertTrue(
    Condition := fb.sts.aFaceplates[4].mapped,
    Message   := 'Faceplate mapped should mirror nActiveMask for that bit');
AssertTrue(
    Condition := fb.sts.aFaceplates[4].bypassable,
    Message   := 'Faceplate bypassable should mirror cfg.nBypassable for that bit');

TEST_FINISHED();
END_METHOD

END_FUNCTION_BLOCK

// ---- Testing/Tests/FB_Interlock_Test.TcPOU
// Integration tests for FB_Interlock on top of FB_BitMatrix64.
// FB_BitMatrix64_Test already covers the shared matrix mechanics, so this
// suite focuses on interlock-specific behaviour:
//   - once a mapped bit goes bad it stays bad (latching), even if the
//     underlying signal recovers on its own
//   - Reset() snaps the latch to the current live value; a still-bad bit
//     stays bad (reset is not a safety override)
//   - unmapped-bad memory keeps bOK FALSE after a bit becomes unmapped
//     while it was bad, and survives until Reset() clears it
//   - bypass still forces a bit good in the effective rollup
//   - Reset() intentionally preserves bypass state
FUNCTION_BLOCK FB_Interlock_Test EXTENDS TcUnit.FB_TestSuite

InitialStateOk();
BadMappedBitLatches();
RecoveryDoesNotClearLatch();
ResetClearsLatchAfterRecovery();
ResetWithActiveBadLeavesItBad();
UnmappedBadMemoryKeepsBOkFalse();
ResetClearsUnmappedBadMemory();
BypassForcesGoodInRollup();
ResetPreservesBypass();

METHOD InitialStateOk
VAR
    fb : TcForge.FB_Interlock;
END_VAR
TEST('InitialStateOk');

fb();

AssertTrue(
    Condition := fb.sts.bOK,
    Message   := 'Fresh interlock with no mappings should report bOK = TRUE');
AssertEquals_ULINT(
    Expected := 16#FFFFFFFFFFFFFFFF,
    Actual   := fb.sts.nInterlocks,
    Message  := 'Fresh interlock rollup should be all-good');
AssertEquals_UDINT(
    Expected := 999,
    Actual   := fb.sts.nFirstFailureBitIndex,
    Message  := 'Fresh interlock should expose the sentinel first-failure index');

TEST_FINISHED();
END_METHOD

METHOD BadMappedBitLatches
VAR
    fb      : TcForge.FB_Interlock;
    bitMask : ULINT;
END_VAR
TEST('BadMappedBitLatches');

bitMask := SHL(ULINT#1, 5);

fb.MapInput(bitIndex := 5, inputValue := FALSE);
fb();

AssertFalse(
    Condition := fb.sts.bOK,
    Message   := 'bOK must be FALSE while bit 5 is bad');
AssertTrue(
    Condition := (fb.sts.nInterlocks AND bitMask) = 0,
    Message   := 'Bit 5 should show as bad in the effective rollup');

TEST_FINISHED();
END_METHOD

METHOD RecoveryDoesNotClearLatch
VAR
    fb : TcForge.FB_Interlock;
END_VAR
TEST('RecoveryDoesNotClearLatch');

// This is the defining interlock behaviour: once bad, stays bad until
// Reset() is explicitly called, even after the input recovers on its own.
fb.MapInput(bitIndex := 5, inputValue := FALSE);
fb();

AssertFalse(
    Condition := fb.sts.bOK,
    Message   := 'Precondition: bOK should be FALSE while bit 5 is bad');

fb.MapInput(bitIndex := 5, inputValue := TRUE);
fb();
fb.MapInput(bitIndex := 5, inputValue := TRUE);
fb();

AssertFalse(
    Condition := fb.sts.bOK,
    Message   := 'Interlock must stay latched FALSE after the input recovers until Reset() is called');

TEST_FINISHED();
END_METHOD

METHOD ResetClearsLatchAfterRecovery
VAR
    fb : TcForge.FB_Interlock;
END_VAR
TEST('ResetClearsLatchAfterRecovery');

// Fault -> recover -> Reset() -> bOK TRUE.
fb.MapInput(bitIndex := 5, inputValue := FALSE);
fb();
fb.MapInput(bitIndex := 5, inputValue := TRUE);
fb();

fb.Reset();
fb.MapInput(bitIndex := 5, inputValue := TRUE);
fb();

AssertTrue(
    Condition := fb.sts.bOK,
    Message   := 'Reset() after recovery must clear the latch and restore bOK = TRUE');

TEST_FINISHED();
END_METHOD

METHOD ResetWithActiveBadLeavesItBad
VAR
    fb : TcForge.FB_Interlock;
END_VAR
TEST('ResetWithActiveBadLeavesItBad');

// Reset() is a latch clear, not a safety override. If the live condition
// is still bad when Reset() is called, bOK must stay FALSE.
fb.MapInput(bitIndex := 5, inputValue := FALSE);
fb();

fb.Reset();
fb.MapInput(bitIndex := 5, inputValue := FALSE);
fb();

AssertFalse(
    Condition := fb.sts.bOK,
    Message   := 'Reset() while the condition is still bad must NOT clear the failure');

TEST_FINISHED();
END_METHOD

METHOD UnmappedBadMemoryKeepsBOkFalse
VAR
    fb : TcForge.FB_Interlock;
    i  : UDINT;
END_VAR
TEST('UnmappedBadMemoryKeepsBOkFalse');

// Map bit 5 as bad exactly once, then stop feeding. After MAPPING_TIMEOUT
// the bit is removed from the active mask — but the interlock must
// remember it was bad at the moment of unmap and keep bOK FALSE until
// Reset() is called. This is the key safety invariant that survived the
// FB_BitMatrix64 extraction.
fb.MapInput(bitIndex := 5, inputValue := FALSE);
fb();

FOR i := 1 TO 15 DO
    fb();
END_FOR;

AssertFalse(
    Condition := fb.sts.bOK,
    Message   := 'Interlock must stay FALSE after a bit became unmapped while bad');

TEST_FINISHED();
END_METHOD

METHOD ResetClearsUnmappedBadMemory
VAR
    fb : TcForge.FB_Interlock;
    i  : UDINT;
END_VAR
TEST('ResetClearsUnmappedBadMemory');

fb.MapInput(bitIndex := 5, inputValue := FALSE);
fb();
FOR i := 1 TO 15 DO
    fb();
END_FOR;

AssertFalse(
    Condition := fb.sts.bOK,
    Message   := 'Precondition: unmapped-bad memory should be holding bOK FALSE');

fb.Reset();
fb();

AssertTrue(
    Condition := fb.sts.bOK,
    Message   := 'Reset() must clear the unmapped-bad memory and restore bOK = TRUE');

TEST_FINISHED();
END_METHOD

METHOD BypassForcesGoodInRollup
VAR
    fb       : TcForge.FB_Interlock;
    bitMask  : ULINT;
    response : TcForge.E_RpcMethodResponse;
END_VAR
TEST('BypassForcesGoodInRollup');

bitMask := SHL(ULINT#1, 5);
fb.cfg.nBypassable := bitMask;

fb.MapInput(bitIndex := 5, inputValue := FALSE);
response := fb.SetBypass(bitIndex := 5, bEnable := TRUE);
fb();

AssertEquals_DINT(
    Expected := TcForge.E_RpcMethodResponse.ACCEPTED,
    Actual   := response,
    Message  := 'SetBypass should accept when the bit is flagged bypassable in cfg');
AssertTrue(
    Condition := fb.sts.bOK,
    Message   := 'A bypassed bit must be forced good in the effective rollup');

TEST_FINISHED();
END_METHOD

METHOD ResetPreservesBypass
VAR
    fb      : TcForge.FB_Interlock;
    bitMask : ULINT;
END_VAR
TEST('ResetPreservesBypass');

bitMask := SHL(ULINT#1, 5);
fb.cfg.nBypassable := bitMask;

fb.SetBypass(bitIndex := 5, bEnable := TRUE);
fb();

AssertTrue(
    Condition := (fb.sts.nBypassMask AND bitMask) <> 0,
    Message   := 'Precondition: bit 5 bypass should be active before Reset()');

fb.Reset();
fb();

AssertTrue(
    Condition := (fb.sts.nBypassMask AND bitMask) <> 0,
    Message   := 'Reset() on an interlock must PRESERVE bypass state (per the public contract)');

TEST_FINISHED();
END_METHOD

END_FUNCTION_BLOCK

// ---- Testing/Tests/FB_AlarmSimple_Test.TcPOU
// FB_AlarmSimple is the thinnest concrete child of FB_AlarmBase, so this
// suite doubles as the test harness for the shared alarm contract:
// enable gating, raw -> active rollup, latch + ack state machine, severity
// propagation, message echo, source-lock gating on Ack().
//
// Debounce (TON/TOF) is intentionally exercised with T#0MS delays; the
// debounce primitive itself is IEC standard and testing its timing under
// TcUnit is awkward because a suite body runs once per task cycle. Every
// test below therefore lets tOnDelay / tOffDelay stay at zero and focuses
// on the alarm logic that sits on top of the debounced signal.
FUNCTION_BLOCK FB_AlarmSimple_Test EXTENDS TcUnit.FB_TestSuite

DisabledSuppressesEverything();
SelfClearingTracksInput();
LatchingHoldsAfterClearWithoutAck();
AckAfterClearReleasesLatch();
AckWhileActiveFlipsAckedButNotLatch();
SeverityFollowsActiveState();
MessageEchoedFromCfg();
DisableClearsActiveLatch();
LockedSourceRejectsOperatorAck();
AckWithNoLatchIsNoOp();

METHOD DisabledSuppressesEverything
VAR
    fb : TcForge.FB_AlarmSimple;
END_VAR
TEST('DisabledSuppressesEverything');

// cfg.bEnable defaults to FALSE; even with the input firing, the alarm
// must stay inert and report severity NONE.
fb.cfg.common.eSeverity := TcForge.E_AlarmSeverity.CRITICAL;

fb(inpActive := TRUE);

AssertFalse(
    Condition := fb.sts.active,
    Message   := 'Disabled alarm must not go active');
AssertEquals_USINT(
    Expected := TcForge.E_AlarmSeverity.NONE,
    Actual   := fb.sts.eSeverity,
    Message  := 'Disabled alarm must report severity NONE');

TEST_FINISHED();
END_METHOD

METHOD SelfClearingTracksInput
VAR
    fb : TcForge.FB_AlarmSimple;
END_VAR
TEST('SelfClearingTracksInput');

// bRequireAck = FALSE => no latch. active follows the debounced input
// in both directions.
fb.cfg.common.bEnable     := TRUE;
fb.cfg.common.bRequireAck := FALSE;
fb.cfg.common.eSeverity   := TcForge.E_AlarmSeverity.WARNING;

fb(inpActive := TRUE);
AssertTrue(
    Condition := fb.sts.active,
    Message   := 'Non-latching alarm should go active when the input is TRUE');

fb(inpActive := FALSE);
AssertFalse(
    Condition := fb.sts.active,
    Message   := 'Non-latching alarm should clear the same cycle the input clears');
AssertFalse(
    Condition := fb.sts.latched,
    Message   := 'Non-latching alarm must never expose latched');

TEST_FINISHED();
END_METHOD

METHOD LatchingHoldsAfterClearWithoutAck
VAR
    fb : TcForge.FB_AlarmSimple;
END_VAR
TEST('LatchingHoldsAfterClearWithoutAck');

fb.cfg.common.bEnable     := TRUE;
fb.cfg.common.bRequireAck := TRUE;
fb.cfg.common.eSeverity   := TcForge.E_AlarmSeverity.CRITICAL;

fb(inpActive := TRUE);
AssertTrue(
    Condition := fb.sts.active,
    Message   := 'Latching alarm should go active when the input fires');
AssertTrue(
    Condition := fb.sts.latched,
    Message   := 'latched should indicate an un-acked latch');

fb(inpActive := FALSE);
AssertTrue(
    Condition := fb.sts.active,
    Message   := 'Latching alarm must stay active after the input clears until Ack()');

TEST_FINISHED();
END_METHOD

METHOD AckAfterClearReleasesLatch
VAR
    fb       : TcForge.FB_AlarmSimple;
    response : TcForge.E_RpcMethodResponse;
END_VAR
TEST('AckAfterClearReleasesLatch');

fb.cfg.common.bEnable     := TRUE;
fb.cfg.common.bRequireAck := TRUE;
fb.cfg.common.eSeverity   := TcForge.E_AlarmSeverity.WARNING;

// Trip, clear the condition, then ack — latch should release next cycle.
fb(inpActive := TRUE);
fb(inpActive := FALSE);

response := fb.Ack(eRequester := TcForge.E_Requester.OPERATOR);
fb(inpActive := FALSE);

AssertEquals_DINT(
    Expected := TcForge.E_RpcMethodResponse.ACCEPTED,
    Actual   := response,
    Message  := 'Ack() with no source lock should be accepted');
AssertFalse(
    Condition := fb.sts.active,
    Message   := 'Latch must release once condition has cleared AND Ack() has been called');

TEST_FINISHED();
END_METHOD

METHOD AckWhileActiveFlipsAckedButNotLatch
VAR
    fb : TcForge.FB_AlarmSimple;
END_VAR
TEST('AckWhileActiveFlipsAckedButNotLatch');

fb.cfg.common.bEnable     := TRUE;
fb.cfg.common.bRequireAck := TRUE;
fb.cfg.common.eSeverity   := TcForge.E_AlarmSeverity.CRITICAL;

// Condition still firing when the operator acks — valid middle state:
// active stays TRUE, acked becomes TRUE, latched becomes FALSE
// (operator has seen it but the process is still in the bad state).
fb(inpActive := TRUE);
fb.Ack(eRequester := TcForge.E_Requester.OPERATOR);
fb(inpActive := TRUE);

AssertTrue(
    Condition := fb.sts.active,
    Message   := 'active should remain TRUE while the condition is still firing');
AssertTrue(
    Condition := fb.sts.acked,
    Message   := 'acked should be TRUE after an accepted Ack()');
AssertFalse(
    Condition := fb.sts.latched,
    Message   := 'latched should drop once the latch has been acknowledged');

TEST_FINISHED();
END_METHOD

METHOD SeverityFollowsActiveState
VAR
    fb : TcForge.FB_AlarmSimple;
END_VAR
TEST('SeverityFollowsActiveState');

fb.cfg.common.bEnable     := TRUE;
fb.cfg.common.bRequireAck := FALSE;
fb.cfg.common.eSeverity   := TcForge.E_AlarmSeverity.CRITICAL;

fb(inpActive := TRUE);
AssertEquals_USINT(
    Expected := TcForge.E_AlarmSeverity.CRITICAL,
    Actual   := fb.sts.eSeverity,
    Message  := 'Active alarm must publish the configured severity');

fb(inpActive := FALSE);
AssertEquals_USINT(
    Expected := TcForge.E_AlarmSeverity.NONE,
    Actual   := fb.sts.eSeverity,
    Message  := 'Inactive alarm must publish severity NONE (aggregators MAX() across alarms)');

TEST_FINISHED();
END_METHOD

METHOD MessageEchoedFromCfg
VAR
    fb : TcForge.FB_AlarmSimple;
END_VAR
TEST('MessageEchoedFromCfg');

fb.cfg.common.bEnable  := TRUE;
fb.cfg.common.sMessage := 'Cell door open';

fb(inpActive := FALSE);

AssertEquals_STRING(
    Expected := 'Cell door open',
    Actual   := fb.sts.sMessage,
    Message  := 'sts.sMessage must echo cfg.common.sMessage');

TEST_FINISHED();
END_METHOD

METHOD DisableClearsActiveLatch
VAR
    fb : TcForge.FB_AlarmSimple;
END_VAR
TEST('DisableClearsActiveLatch');

fb.cfg.common.bEnable     := TRUE;
fb.cfg.common.bRequireAck := TRUE;
fb.cfg.common.eSeverity   := TcForge.E_AlarmSeverity.CRITICAL;

// Latch, then disable. Flipping bEnable FALSE must force the alarm inert
// immediately — operator disables dominate any held latch.
fb(inpActive := TRUE);
AssertTrue(
    Condition := fb.sts.active,
    Message   := 'Precondition: latch should be active before disable');

fb.cfg.common.bEnable := FALSE;
fb(inpActive := TRUE);

AssertFalse(
    Condition := fb.sts.active,
    Message   := 'Disable must drop active even while the input is still firing');
AssertFalse(
    Condition := fb.sts.latched,
    Message   := 'Disable must clear latched');
AssertEquals_USINT(
    Expected := TcForge.E_AlarmSeverity.NONE,
    Actual   := fb.sts.eSeverity,
    Message  := 'Disable must drop severity back to NONE');

TEST_FINISHED();
END_METHOD

METHOD LockedSourceRejectsOperatorAck
VAR
    fb        : TcForge.FB_AlarmSimple;
    opResp    : TcForge.E_RpcMethodResponse;
    progResp  : TcForge.E_RpcMethodResponse;
END_VAR
TEST('LockedSourceRejectsOperatorAck');

fb.cfg.common.bEnable     := TRUE;
fb.cfg.common.bRequireAck := TRUE;
fb.cfg.common.eSeverity   := TcForge.E_AlarmSeverity.CRITICAL;

fb.LockSource(bLock := TRUE);
fb(inpActive := TRUE);

opResp   := fb.Ack(eRequester := TcForge.E_Requester.OPERATOR);
progResp := fb.Ack(eRequester := TcForge.E_Requester.PROG);

AssertEquals_DINT(
    Expected := TcForge.E_RpcMethodResponse.REJECTED_SOURCE_NOT_ALLOWED,
    Actual   := opResp,
    Message  := 'Source-locked alarm must reject OPERATOR Ack()');
AssertEquals_DINT(
    Expected := TcForge.E_RpcMethodResponse.ACCEPTED,
    Actual   := progResp,
    Message  := 'Source-locked alarm must still accept PROG Ack()');

TEST_FINISHED();
END_METHOD

METHOD AckWithNoLatchIsNoOp
VAR
    fb       : TcForge.FB_AlarmSimple;
    response : TcForge.E_RpcMethodResponse;
END_VAR
TEST('AckWithNoLatchIsNoOp');

fb.cfg.common.bEnable     := TRUE;
fb.cfg.common.bRequireAck := TRUE;

// Ack() before any latch exists is accepted (the requester validation
// passes) but must leave acked FALSE — there is nothing to mark acked.
fb(inpActive := FALSE);
response := fb.Ack(eRequester := TcForge.E_Requester.OPERATOR);
fb(inpActive := FALSE);

AssertEquals_DINT(
    Expected := TcForge.E_RpcMethodResponse.ACCEPTED,
    Actual   := response,
    Message  := 'Ack() with no latch returns ACCEPTED (validation passes)');
AssertFalse(
    Condition := fb.sts.acked,
    Message   := 'Ack() with no latch must NOT flip acked — there is no latch to ack');

TEST_FINISHED();
END_METHOD

END_FUNCTION_BLOCK

// ---- Testing/Tests/FB_AlarmLimit_Test.TcPOU
// Tests for FB_AlarmLimit — four-level (HiHi/Hi/Lo/LoLo) ladder built by
// composing FB_AlarmThreshold. FB_AlarmSimple_Test already covers the
// shared FB_AlarmBase contract, so this suite focuses on the composite
// behaviour that lives only here:
//   - per-direction threshold evaluation via bFailHigh / bFailLow
//   - flood suppression (HiHi hides Hi, LoLo hides Lo) on the rollup flags
//     while keeping the raw sub-statuses available
//   - severity aggregation (highest-active wins)
//   - anyActive is the OR of all four rollup flags
//   - Ack() cascades to every level
FUNCTION_BLOCK FB_AlarmLimit_Test EXTENDS TcUnit.FB_TestSuite

AllDisabledStaysSilent();
HiTripsAboveThreshold();
HiHiSuppressesHiOnRollup();
LoTripsBelowThreshold();
LoLoSuppressesLoOnRollup();
SeverityIsHighestActiveLevel();
AnyActiveReflectsRollup();
AckCascadesToEveryLevel();

// Helper: configure HiHi and Hi as a typical upper ladder. Keeps each
// test method short and consistent with the example PRG_Alarms wiring.
METHOD PRIVATE _ConfigureHiHi
VAR_IN_OUT
    fb : TcForge.FB_AlarmLimit;
END_VAR
fb.cfg.HiHi.common.bEnable     := TRUE;
fb.cfg.HiHi.common.bRequireAck := FALSE;
fb.cfg.HiHi.common.eSeverity   := TcForge.E_AlarmSeverity.CRITICAL;
fb.cfg.HiHi.fThreshold         := 110.0;
fb.cfg.HiHi.bFailHigh          := TRUE;

fb.cfg.Hi.common.bEnable     := TRUE;
fb.cfg.Hi.common.bRequireAck := FALSE;
fb.cfg.Hi.common.eSeverity   := TcForge.E_AlarmSeverity.WARNING;
fb.cfg.Hi.fThreshold         := 100.0;
fb.cfg.Hi.bFailHigh          := TRUE;
END_METHOD

// Helper: configure Lo and LoLo as a typical lower ladder.
METHOD PRIVATE _ConfigureLoLo
VAR_IN_OUT
    fb : TcForge.FB_AlarmLimit;
END_VAR
fb.cfg.Lo.common.bEnable     := TRUE;
fb.cfg.Lo.common.bRequireAck := FALSE;
fb.cfg.Lo.common.eSeverity   := TcForge.E_AlarmSeverity.WARNING;
fb.cfg.Lo.fThreshold         := 20.0;
fb.cfg.Lo.bFailLow           := TRUE;

fb.cfg.LoLo.common.bEnable     := TRUE;
fb.cfg.LoLo.common.bRequireAck := FALSE;
fb.cfg.LoLo.common.eSeverity   := TcForge.E_AlarmSeverity.CRITICAL;
fb.cfg.LoLo.fThreshold         := 10.0;
fb.cfg.LoLo.bFailLow           := TRUE;
END_METHOD

METHOD AllDisabledStaysSilent
VAR
    fb : TcForge.FB_AlarmLimit;
END_VAR
TEST('AllDisabledStaysSilent');

// Every level disabled; rollup flags and severity must stay quiet even
// when the process value is far outside every sensible band.
fb(inpPv := 500.0);

AssertFalse(
    Condition := fb.sts.anyActive,
    Message   := 'anyActive must be FALSE when every level is disabled');
AssertEquals_USINT(
    Expected := TcForge.E_AlarmSeverity.NONE,
    Actual   := fb.sts.eSeverity,
    Message  := 'eSeverity must be NONE when every level is disabled');

TEST_FINISHED();
END_METHOD

METHOD HiTripsAboveThreshold
VAR
    fb : TcForge.FB_AlarmLimit;
END_VAR
TEST('HiTripsAboveThreshold');

_ConfigureHiHi(fb := fb);

fb(inpPv := 105.0);  // above Hi (100), below HiHi (110)

AssertTrue(
    Condition := fb.sts.hiActive,
    Message   := 'Hi should trip when PV crosses its threshold');
AssertFalse(
    Condition := fb.sts.hiHiActive,
    Message   := 'HiHi should stay inactive while PV is below the HiHi threshold');

TEST_FINISHED();
END_METHOD

METHOD HiHiSuppressesHiOnRollup
VAR
    fb : TcForge.FB_AlarmLimit;
END_VAR
TEST('HiHiSuppressesHiOnRollup');

_ConfigureHiHi(fb := fb);

fb(inpPv := 115.0);  // above both Hi and HiHi

AssertTrue(
    Condition := fb.sts.hiHiActive,
    Message   := 'HiHi should trip when PV crosses its threshold');
AssertFalse(
    Condition := fb.sts.hiActive,
    Message   := 'Hi must be suppressed on the rollup while HiHi is active');
AssertTrue(
    Condition := fb.sts.Hi.active,
    Message   := 'Raw Hi sub-status must still expose the trip (forensics channel)');

TEST_FINISHED();
END_METHOD

METHOD LoTripsBelowThreshold
VAR
    fb : TcForge.FB_AlarmLimit;
END_VAR
TEST('LoTripsBelowThreshold');

_ConfigureLoLo(fb := fb);

fb(inpPv := 15.0);  // below Lo (20), above LoLo (10)

AssertTrue(
    Condition := fb.sts.loActive,
    Message   := 'Lo should trip when PV drops below its threshold');
AssertFalse(
    Condition := fb.sts.loLoActive,
    Message   := 'LoLo should stay inactive while PV is above the LoLo threshold');

TEST_FINISHED();
END_METHOD

METHOD LoLoSuppressesLoOnRollup
VAR
    fb : TcForge.FB_AlarmLimit;
END_VAR
TEST('LoLoSuppressesLoOnRollup');

_ConfigureLoLo(fb := fb);

fb(inpPv := 5.0);  // below both Lo and LoLo

AssertTrue(
    Condition := fb.sts.loLoActive,
    Message   := 'LoLo should trip when PV drops below its threshold');
AssertFalse(
    Condition := fb.sts.loActive,
    Message   := 'Lo must be suppressed on the rollup while LoLo is active');
AssertTrue(
    Condition := fb.sts.Lo.active,
    Message   := 'Raw Lo sub-status must still expose the trip (forensics channel)');

TEST_FINISHED();
END_METHOD

METHOD SeverityIsHighestActiveLevel
VAR
    fb : TcForge.FB_AlarmLimit;
END_VAR
TEST('SeverityIsHighestActiveLevel');

_ConfigureHiHi(fb := fb);

// PV between Hi and HiHi → only Hi active → severity = WARNING.
fb(inpPv := 105.0);
AssertEquals_USINT(
    Expected := TcForge.E_AlarmSeverity.WARNING,
    Actual   := fb.sts.eSeverity,
    Message  := 'Severity should be WARNING when only Hi is active');

// PV above HiHi → HiHi (CRITICAL) wins even though raw Hi still fires.
fb(inpPv := 115.0);
AssertEquals_USINT(
    Expected := TcForge.E_AlarmSeverity.CRITICAL,
    Actual   := fb.sts.eSeverity,
    Message  := 'Severity should be CRITICAL once HiHi engages');

TEST_FINISHED();
END_METHOD

METHOD AnyActiveReflectsRollup
VAR
    fb : TcForge.FB_AlarmLimit;
END_VAR
TEST('AnyActiveReflectsRollup');

_ConfigureHiHi(fb := fb);
_ConfigureLoLo(fb := fb);

fb(inpPv := 50.0);  // in the good band
AssertFalse(
    Condition := fb.sts.anyActive,
    Message   := 'anyActive should be FALSE while PV sits in the good band');

fb(inpPv := 115.0);
AssertTrue(
    Condition := fb.sts.anyActive,
    Message   := 'anyActive should be TRUE once any level trips');

fb(inpPv := 50.0);
AssertFalse(
    Condition := fb.sts.anyActive,
    Message   := 'anyActive should go back FALSE when PV returns to the good band (non-latching cfg)');

TEST_FINISHED();
END_METHOD

METHOD AckCascadesToEveryLevel
VAR
    fb       : TcForge.FB_AlarmLimit;
    response : TcForge.E_RpcMethodResponse;
END_VAR
TEST('AckCascadesToEveryLevel');

// Both Hi and HiHi latching — a PV spike into HiHi latches both raw
// sub-alarms. Ack() must cascade so every level releases on the next
// post-clear cycle.
fb.cfg.HiHi.common.bEnable     := TRUE;
fb.cfg.HiHi.common.bRequireAck := TRUE;
fb.cfg.HiHi.common.eSeverity   := TcForge.E_AlarmSeverity.CRITICAL;
fb.cfg.HiHi.fThreshold         := 110.0;
fb.cfg.HiHi.bFailHigh          := TRUE;

fb.cfg.Hi.common.bEnable     := TRUE;
fb.cfg.Hi.common.bRequireAck := TRUE;
fb.cfg.Hi.common.eSeverity   := TcForge.E_AlarmSeverity.WARNING;
fb.cfg.Hi.fThreshold         := 100.0;
fb.cfg.Hi.bFailHigh          := TRUE;

// Spike then recover.
fb(inpPv := 115.0);
fb(inpPv := 50.0);

AssertTrue(
    Condition := fb.sts.HiHi.active AND fb.sts.Hi.active,
    Message   := 'Precondition: both raw sub-alarms should be latched after the spike');

response := fb.Ack(eRequester := TcForge.E_Requester.OPERATOR);
fb(inpPv := 50.0);

AssertEquals_DINT(
    Expected := TcForge.E_RpcMethodResponse.ACCEPTED,
    Actual   := response,
    Message  := 'Composite Ack() should be accepted when at least one level accepts');
AssertFalse(
    Condition := fb.sts.HiHi.active,
    Message   := 'HiHi latch must release after cascaded Ack() + clear');
AssertFalse(
    Condition := fb.sts.Hi.active,
    Message   := 'Hi latch must release after cascaded Ack() + clear');
AssertFalse(
    Condition := fb.sts.anyActive,
    Message   := 'anyActive should return FALSE once every level releases');

TEST_FINISHED();
END_METHOD

END_FUNCTION_BLOCK

// ---- Testing/Tests/FB_DeviceBase_Test.TcPOU
// Tests for FB_DeviceBase — the shared base for every TcForge device FB.
// Driven through FB_DeviceBase_Probe (a test-only concrete child) because
// the base is ABSTRACT and the fault book-keeping API is PROTECTED.
//
// Coverage focuses on the contract every device inherits:
//   - diagnostics (IsFaulted / GetFaultCode / GetFaultString with virtual
//     dispatch through the child's ResolveFaultString)
//   - _Raise semantics: zero-code no-op, idempotent on code within an
//     episode, different code replaces the active fault
//   - _ClearFault wipes the active fault but preserves lastFault* for
//     the header so HMIs can still render what happened
//   - Reset() is always accepted from any requester — safety invariant
//   - _UpdateHeader() mirrors the active/last fault, source-lock, busy,
//     and ready state into ST_DeviceHeader_Sts
//   - LockSource() makes sourceLocked and forces ready FALSE
FUNCTION_BLOCK FB_DeviceBase_Test EXTENDS TcUnit.FB_TestSuite

FreshInstanceNotFaulted();
RaiseZeroCodeIsNoOp();
RaiseSetsActiveFaultAndResolvesString();
RaiseSameCodeIsIdempotent();
DifferentCodeReplacesActiveFault();
ClearFaultWipesActiveButKeepsLastFault();
ResetAlwaysAcceptedEvenFromOperatorWhileLocked();
HeaderMirrorsActiveFault();
HeaderReadyGoesFalseOnSourceLock();
HeaderReadyGoesFalseOnBusy();

METHOD FreshInstanceNotFaulted
VAR
    fb : FB_DeviceBase_Probe;
END_VAR
TEST('FreshInstanceNotFaulted');

AssertFalse(
    Condition := fb.IsFaulted(),
    Message   := 'Fresh device must not be faulted');
AssertEquals_DINT(
    Expected := 0,
    Actual   := fb.GetFaultCode(),
    Message  := 'Fresh device fault code should be 0');
AssertEquals_STRING(
    Expected := '',
    Actual   := fb.GetFaultString(),
    Message  := 'Fresh device fault string should be empty');

TEST_FINISHED();
END_METHOD

METHOD RaiseZeroCodeIsNoOp
VAR
    fb     : FB_DeviceBase_Probe;
    result : BOOL;
END_VAR
TEST('RaiseZeroCodeIsNoOp');

// code = 0 is the "no fault" sentinel; calling _Raise(0, ...) must never
// register a fault nor push a ring entry.
result := fb.ProbeRaise(code := 0, source := 'test', reason := 'should not register');

AssertFalse(
    Condition := result,
    Message   := '_Raise(0) must return FALSE (nothing was pushed)');
AssertFalse(
    Condition := fb.IsFaulted(),
    Message   := '_Raise(0) must not put the device into a faulted state');

TEST_FINISHED();
END_METHOD

METHOD RaiseSetsActiveFaultAndResolvesString
VAR
    fb     : FB_DeviceBase_Probe;
    result : BOOL;
END_VAR
TEST('RaiseSetsActiveFaultAndResolvesString');

result := fb.ProbeRaise(code := 42, source := 'step5', reason := 'motion timeout');

AssertTrue(
    Condition := result,
    Message   := '_Raise of a new non-zero code must return TRUE (ring entry pushed)');
AssertTrue(
    Condition := fb.IsFaulted(),
    Message   := 'IsFaulted should be TRUE after a raise');
AssertEquals_DINT(
    Expected := 42,
    Actual   := fb.GetFaultCode(),
    Message  := 'GetFaultCode should report the raised code');
AssertEquals_STRING(
    Expected := 'Motion timeout',
    Actual   := fb.GetFaultString(),
    Message  := 'GetFaultString should resolve via the child ResolveFaultString override');

TEST_FINISHED();
END_METHOD

METHOD RaiseSameCodeIsIdempotent
VAR
    fb         : FB_DeviceBase_Probe;
    firstCall  : BOOL;
    secondCall : BOOL;
END_VAR
TEST('RaiseSameCodeIsIdempotent');

// Cyclic callers often raise the same fault every scan until cleared.
// A second raise of the same non-zero code within one episode must be a
// no-op so the ring buffer doesn't flood.
firstCall  := fb.ProbeRaise(code := 42, source := 'step5', reason := 'first call');
secondCall := fb.ProbeRaise(code := 42, source := 'step5', reason := 'second call — ignored');

AssertTrue(
    Condition := firstCall,
    Message   := 'First _Raise of a code must return TRUE');
AssertFalse(
    Condition := secondCall,
    Message   := 'Repeat _Raise of the same code within an episode must return FALSE (no new ring entry)');
AssertEquals_DINT(
    Expected := 42,
    Actual   := fb.GetFaultCode(),
    Message  := 'Active fault must still be the first code after a repeated raise');

TEST_FINISHED();
END_METHOD

METHOD DifferentCodeReplacesActiveFault
VAR
    fb      : FB_DeviceBase_Probe;
    first   : BOOL;
    second  : BOOL;
END_VAR
TEST('DifferentCodeReplacesActiveFault');

// A progression like 'Timeout' -> 'LimitTripped' should preserve both in
// the ring; the second raise returns TRUE and becomes the active fault.
first  := fb.ProbeRaise(code := 42, source := 'step5', reason := 'motion timeout');
second := fb.ProbeRaise(code := 99, source := 'step5', reason := 'limit tripped');

AssertTrue(
    Condition := first AND second,
    Message   := 'Both raises of different codes must return TRUE');
AssertEquals_DINT(
    Expected := 99,
    Actual   := fb.GetFaultCode(),
    Message  := 'Active fault must be the most recent code');
AssertEquals_STRING(
    Expected := 'Limit tripped',
    Actual   := fb.GetFaultString(),
    Message  := 'GetFaultString must reflect the new active code');

TEST_FINISHED();
END_METHOD

METHOD ClearFaultWipesActiveButKeepsLastFault
VAR
    fb : FB_DeviceBase_Probe;
END_VAR
TEST('ClearFaultWipesActiveButKeepsLastFault');

fb.ProbeRaise(code := 42, source := 'step5', reason := 'motion timeout');
fb.ProbeClearFault();

AssertFalse(
    Condition := fb.IsFaulted(),
    Message   := '_ClearFault must drop IsFaulted to FALSE');
AssertEquals_DINT(
    Expected := 0,
    Actual   := fb.GetFaultCode(),
    Message  := 'Active fault code must be 0 after _ClearFault');

// Header must still preserve last-fault fields so the HMI can render
// "last fault: motion timeout".
fb.Refresh(stateString := 'IDLE', busy := FALSE);

AssertEquals_DINT(
    Expected := 42,
    Actual   := fb.header.lastFaultCode,
    Message  := 'header.lastFaultCode must preserve history after _ClearFault');
AssertEquals_STRING(
    Expected := 'Motion timeout',
    Actual   := fb.header.lastFaultString,
    Message  := 'header.lastFaultString must preserve the resolved text after _ClearFault');

TEST_FINISHED();
END_METHOD

METHOD ResetAlwaysAcceptedEvenFromOperatorWhileLocked
VAR
    fb       : FB_DeviceBase_Probe;
    response : TcForge.E_RpcMethodResponse;
END_VAR
TEST('ResetAlwaysAcceptedEvenFromOperatorWhileLocked');

// Safety invariant: Reset() is always accepted, regardless of source lock
// or active fault. No one should be locked out of clearing a fault.
fb.LockSource(bLock := TRUE);
fb.ProbeRaise(code := 42, source := 'step5', reason := 'motion timeout');

response := fb.Reset(eRequester := TcForge.E_Requester.OPERATOR);

AssertEquals_DINT(
    Expected := TcForge.E_RpcMethodResponse.ACCEPTED,
    Actual   := response,
    Message  := 'Reset() must be accepted from OPERATOR even while source-locked');
AssertFalse(
    Condition := fb.IsFaulted(),
    Message   := 'Reset() must clear the active fault');

TEST_FINISHED();
END_METHOD

METHOD HeaderMirrorsActiveFault
VAR
    fb : FB_DeviceBase_Probe;
END_VAR
TEST('HeaderMirrorsActiveFault');

fb.ProbeRaise(code := 99, source := 'limit_sw', reason := 'upper limit hit');
fb.Refresh(stateString := 'FAULTED', busy := FALSE);

AssertTrue(
    Condition := fb.header.faulted,
    Message   := 'header.faulted must be TRUE while a fault is active');
AssertFalse(
    Condition := fb.header.ready,
    Message   := 'header.ready must be FALSE while faulted');
AssertEquals_DINT(
    Expected := 99,
    Actual   := fb.header.faultCode,
    Message  := 'header.faultCode must mirror the active fault');
AssertEquals_STRING(
    Expected := 'Limit tripped',
    Actual   := fb.header.faultString,
    Message  := 'header.faultString must resolve via the child override');
AssertEquals_STRING(
    Expected := 'limit_sw',
    Actual   := fb.header.faultSource,
    Message  := 'header.faultSource must carry the raise() source');
AssertEquals_STRING(
    Expected := 'upper limit hit',
    Actual   := fb.header.faultReason,
    Message  := 'header.faultReason must carry the raise() reason');
AssertEquals_STRING(
    Expected := 'FAULTED',
    Actual   := fb.header.stateString,
    Message  := 'header.stateString must mirror the state string passed to _UpdateHeader');

TEST_FINISHED();
END_METHOD

METHOD HeaderReadyGoesFalseOnSourceLock
VAR
    fb : FB_DeviceBase_Probe;
END_VAR
TEST('HeaderReadyGoesFalseOnSourceLock');

fb.Refresh(stateString := 'IDLE', busy := FALSE);
AssertTrue(
    Condition := fb.header.ready,
    Message   := 'Precondition: an idle / unlocked / unfaulted device must be ready');

fb.LockSource(bLock := TRUE);
fb.Refresh(stateString := 'IDLE', busy := FALSE);

AssertTrue(
    Condition := fb.header.sourceLocked,
    Message   := 'header.sourceLocked must mirror LockSource(TRUE)');
AssertFalse(
    Condition := fb.header.ready,
    Message   := 'header.ready must be FALSE while source is locked');

TEST_FINISHED();
END_METHOD

METHOD HeaderReadyGoesFalseOnBusy
VAR
    fb : FB_DeviceBase_Probe;
END_VAR
TEST('HeaderReadyGoesFalseOnBusy');

fb.Refresh(stateString := 'MOVING', busy := TRUE);

AssertTrue(
    Condition := fb.header.busy,
    Message   := 'header.busy must mirror the busy flag passed to _UpdateHeader');
AssertFalse(
    Condition := fb.header.ready,
    Message   := 'header.ready must be FALSE while busy');

TEST_FINISHED();
END_METHOD

END_FUNCTION_BLOCK

// ---- Testing/Tests/FB_LPF_FirstOrder_IIR_Test.TcPOU
// Tests for FB_LPF_FirstOrder_IIR — exponential-smoothing low-pass filter.
// Pure math, no external coupling, so each test drives a fresh instance
// with deterministic samples and checks the output against the closed-
// form IIR recurrence:
//     alpha = dt / (tau + dt)
//     y[n]  = y[n-1] + alpha * (x[n] - y[n-1])
//
// Floating-point results are compared with a tolerance via AssertTrue on
// ABS(actual - expected); TcUnit's primitive AssertEquals_LREAL does not
// accept a delta.
FUNCTION_BLOCK FB_LPF_FirstOrder_IIR_Test EXTENDS TcUnit.FB_TestSuite
VAR CONSTANT
    TOL : LREAL := 1E-9;  // generous floating-point tolerance for LREAL math
END_VAR

ZeroDtBypassesFilterAndRaisesError();
ZeroTauBypassesFilterAndRaisesError();
FirstSampleMatchesIirRecurrence();
StateCarriesBetweenCalls();
ConvergesTowardInputOverManySamples();
ErrorClearsOnValidInputAfterBadInput();

METHOD ZeroDtBypassesFilterAndRaisesError
VAR
    fb : TcForge.FB_LPF_FirstOrder_IIR;
END_VAR
TEST('ZeroDtBypassesFilterAndRaisesError');

// dt <= 0 cannot drive the recurrence, so the filter must fall back to
// passthrough and surface bError so the caller can notice.
fb(fInput := 42.0, fDt := 0.0, fTau := 1.0);

AssertTrue(
    Condition := ABS(fb.fOutput - 42.0) < TOL,
    Message   := 'With fDt = 0 the filter must pass the input through unchanged');
AssertTrue(
    Condition := fb.bError,
    Message   := 'With fDt = 0 the filter must raise bError');

TEST_FINISHED();
END_METHOD

METHOD ZeroTauBypassesFilterAndRaisesError
VAR
    fb : TcForge.FB_LPF_FirstOrder_IIR;
END_VAR
TEST('ZeroTauBypassesFilterAndRaisesError');

fb(fInput := 7.5, fDt := 0.1, fTau := 0.0);

AssertTrue(
    Condition := ABS(fb.fOutput - 7.5) < TOL,
    Message   := 'With fTau = 0 the filter must pass the input through unchanged');
AssertTrue(
    Condition := fb.bError,
    Message   := 'With fTau = 0 the filter must raise bError');

TEST_FINISHED();
END_METHOD

METHOD FirstSampleMatchesIirRecurrence
VAR
    fb       : TcForge.FB_LPF_FirstOrder_IIR;
    expected : LREAL;
    alpha    : LREAL;
END_VAR
TEST('FirstSampleMatchesIirRecurrence');

// Fresh instance: _prevOutput_sync = 0. With input 10, dt 0.1, tau 1.0:
//   alpha = 0.1 / 1.1
//   y[0]  = 0 + alpha * (10 - 0) = alpha * 10
alpha    := 0.1 / 1.1;
expected := alpha * 10.0;

fb(fInput := 10.0, fDt := 0.1, fTau := 1.0);

AssertFalse(
    Condition := fb.bError,
    Message   := 'Valid dt / tau must clear bError');
AssertTrue(
    Condition := ABS(fb.fOutput - expected) < TOL,
    Message   := 'First sample must match the IIR recurrence against zero state');

TEST_FINISHED();
END_METHOD

METHOD StateCarriesBetweenCalls
VAR
    fb        : TcForge.FB_LPF_FirstOrder_IIR;
    alpha     : LREAL;
    y1        : LREAL;
    yExpected : LREAL;
END_VAR
TEST('StateCarriesBetweenCalls');

alpha := 0.1 / 1.1;

fb(fInput := 10.0, fDt := 0.1, fTau := 1.0);
y1 := fb.fOutput;

// Second sample: y[1] = y[0] + alpha * (10 - y[0])
yExpected := y1 + alpha * (10.0 - y1);

fb(fInput := 10.0, fDt := 0.1, fTau := 1.0);

AssertTrue(
    Condition := ABS(fb.fOutput - yExpected) < TOL,
    Message   := 'Second sample must fold the previous output through the IIR recurrence (state is preserved across calls)');

TEST_FINISHED();
END_METHOD

METHOD ConvergesTowardInputOverManySamples
VAR
    fb     : TcForge.FB_LPF_FirstOrder_IIR;
    target : LREAL := 10.0;
    i      : UDINT;
END_VAR
TEST('ConvergesTowardInputOverManySamples');

// 200 samples at dt = tau/20 is well past steady-state — the output must
// be within ~1e-3 of the input regardless of the exact alpha value.
FOR i := 1 TO 200 DO
    fb(fInput := target, fDt := 0.05, fTau := 1.0);
END_FOR;

AssertTrue(
    Condition := ABS(fb.fOutput - target) < 1E-3,
    Message   := 'After many samples the filter output must converge toward the input');

TEST_FINISHED();
END_METHOD

METHOD ErrorClearsOnValidInputAfterBadInput
VAR
    fb : TcForge.FB_LPF_FirstOrder_IIR;
END_VAR
TEST('ErrorClearsOnValidInputAfterBadInput');

// A bad sample raises the flag; the very next valid sample must clear it.
fb(fInput := 5.0, fDt := 0.0, fTau := 1.0);
AssertTrue(
    Condition := fb.bError,
    Message   := 'Precondition: bError should be TRUE after a bad sample');

fb(fInput := 5.0, fDt := 0.1, fTau := 1.0);
AssertFalse(
    Condition := fb.bError,
    Message   := 'bError must clear the cycle a valid sample lands');

TEST_FINISHED();
END_METHOD

END_FUNCTION_BLOCK

// ---- Testing/Tests/FB_DigitalOutput_Test.TcPOU
// Tests for FB_DigitalOutput. Focus is on the behavior the device exposes
// to callers and HMIs:
//
//   * command routing through F_ValidateRequester (source lock)
//   * request-vs-output bookkeeping (commanded always reflects the
//     latest intent, value always reflects the physical bit)
//   * debounce timers actually gating the output
//   * invert in Regular mode
//   * BAD quality holding the last-known-good output
//   * edge pulses being exactly one scan wide
//   * SinglePulse arming on rising edge and cancelling on commanded LOW
//
// Time-dependent behavior is covered by choosing timer values that either
// clamp to zero (instant fire) or stay effectively infinite for the test
// (T#1S), so a single cyclic call lands in the branch under test without
// waiting real time.
FUNCTION_BLOCK FB_DigitalOutput_Test EXTENDS TcUnit.FB_TestSuite

InitialStateReady();
SetOnFromProgDrivesOutputHigh();
SetOffAfterSetOnDrivesOutputLow();
SetOnAcceptedFromProgEvenWhenLocked();
SetOnRejectedFromOperatorWhenLocked();
DebounceOnBlocksOutputUntilElapsed();
DebounceOffHoldsOutputHighUntilElapsed();
InvertFlipsOutputInRegularMode();
BadQualityHoldsLastKnownGoodOutput();
StsCommandedMirrorsRequestEvenUnderBadQuality();
EdgePulsesAreOneScanWide();
SinglePulseFiresOnCommandAndCanBeCanceled();

METHOD InitialStateReady
VAR
    fb : TcForge.FB_DigitalOutput;
END_VAR
TEST('InitialStateReady');

// Fresh instance + one good-quality cycle: no commands issued, no faults
// raised, output dead.
fb(inpQuality := TcForge.E_IO_Quality.GOOD);

AssertFalse(
    Condition := fb.sts.value,
    Message   := 'Fresh instance must start with physical output LOW');
AssertFalse(
    Condition := fb.sts.commanded,
    Message   := 'Fresh instance must start with commanded request LOW');
AssertFalse(
    Condition := fb.sts.header.faulted,
    Message   := 'Fresh instance must not be faulted');
AssertTrue(
    Condition := fb.sts.header.ready,
    Message   := 'Fresh instance must report ready TRUE (no fault, not busy, not locked)');
AssertFalse(
    Condition := fb.sts.header.sourceLocked,
    Message   := 'Fresh instance must not be source-locked');

TEST_FINISHED();
END_METHOD

METHOD SetOnFromProgDrivesOutputHigh
VAR
    fb     : TcForge.FB_DigitalOutput;
    resp   : TcForge.E_RpcMethodResponse;
END_VAR
TEST('SetOnFromProgDrivesOutputHigh');

// Default cfg: no debounce (PT = T#0MS), Regular mode, no invert.
// A single SetOn + one cycle should flush straight through to the
// physical output.
resp := fb.SetOn(eRequester := TcForge.E_Requester.PROG);
fb(inpQuality := TcForge.E_IO_Quality.GOOD);

AssertEquals_DINT(
    Expected := TcForge.E_RpcMethodResponse.ACCEPTED,
    Actual   := resp,
    Message  := 'SetOn from PROG on a fresh instance must be ACCEPTED');
AssertTrue(
    Condition := fb.sts.value,
    Message   := 'Regular mode with no debounce must flush SetOn to the physical output in one cycle');
AssertTrue(
    Condition := fb.sts.commanded,
    Message   := 'commanded must reflect the accepted SetOn request');

TEST_FINISHED();
END_METHOD

METHOD SetOffAfterSetOnDrivesOutputLow
VAR
    fb   : TcForge.FB_DigitalOutput;
    resp : TcForge.E_RpcMethodResponse;
END_VAR
TEST('SetOffAfterSetOnDrivesOutputLow');

fb.SetOn(eRequester := TcForge.E_Requester.PROG);
fb(inpQuality := TcForge.E_IO_Quality.GOOD);

resp := fb.SetOff(eRequester := TcForge.E_Requester.PROG);
fb(inpQuality := TcForge.E_IO_Quality.GOOD);

AssertEquals_DINT(
    Expected := TcForge.E_RpcMethodResponse.ACCEPTED,
    Actual   := resp,
    Message  := 'SetOff from PROG must be ACCEPTED');
AssertFalse(
    Condition := fb.sts.value,
    Message   := 'SetOff must drop the physical output LOW in one cycle with no debounce');
AssertFalse(
    Condition := fb.sts.commanded,
    Message   := 'commanded must follow the latest SetOff request');

TEST_FINISHED();
END_METHOD

METHOD SetOnAcceptedFromProgEvenWhenLocked
VAR
    fb   : TcForge.FB_DigitalOutput;
    resp : TcForge.E_RpcMethodResponse;
END_VAR
TEST('SetOnAcceptedFromProgEvenWhenLocked');

// bSourceLockedToProg is meant to gate OPERATOR; PROG must always get
// through so the program can still drive the output after locking out the
// operator.
fb.LockSource(bLock := TRUE);
resp := fb.SetOn(eRequester := TcForge.E_Requester.PROG);
fb(inpQuality := TcForge.E_IO_Quality.GOOD);

AssertEquals_DINT(
    Expected := TcForge.E_RpcMethodResponse.ACCEPTED,
    Actual   := resp,
    Message  := 'PROG requester must be accepted even with source-lock active');
AssertTrue(
    Condition := fb.sts.value,
    Message   := 'Accepted SetOn from PROG must still drive the physical output');
AssertTrue(
    Condition := fb.sts.header.sourceLocked,
    Message   := 'header must reflect source-lock state');

TEST_FINISHED();
END_METHOD

METHOD SetOnRejectedFromOperatorWhenLocked
VAR
    fb   : TcForge.FB_DigitalOutput;
    resp : TcForge.E_RpcMethodResponse;
END_VAR
TEST('SetOnRejectedFromOperatorWhenLocked');

fb.LockSource(bLock := TRUE);
resp := fb.SetOn(eRequester := TcForge.E_Requester.OPERATOR);
fb(inpQuality := TcForge.E_IO_Quality.GOOD);

AssertEquals_DINT(
    Expected := TcForge.E_RpcMethodResponse.REJECTED_SOURCE_NOT_ALLOWED,
    Actual   := resp,
    Message  := 'OPERATOR requester must be rejected while source-locked');
AssertFalse(
    Condition := fb.sts.value,
    Message   := 'Rejected SetOn must not touch the physical output');
AssertFalse(
    Condition := fb.sts.commanded,
    Message   := 'Rejected SetOn must not update commanded');

TEST_FINISHED();
END_METHOD

METHOD DebounceOnBlocksOutputUntilElapsed
VAR
    fb : TcForge.FB_DigitalOutput;
END_VAR
TEST('DebounceOnBlocksOutputUntilElapsed');

// debounceOn = T#1S — far longer than this synchronous test will run,
// so _tonOn.Q must still be FALSE when we check: the output must be held
// LOW while the debounce hasn't elapsed.
fb.cfg.debounceOn := T#1S;
fb.SetOn(eRequester := TcForge.E_Requester.PROG);
fb(inpQuality := TcForge.E_IO_Quality.GOOD);

AssertTrue(
    Condition := fb.sts.commanded,
    Message   := 'commanded must reflect the request immediately (debounce gates the output, not the request)');
AssertFalse(
    Condition := fb.sts.value,
    Message   := 'debounceOn must hold the physical output LOW until the TON elapses');

TEST_FINISHED();
END_METHOD

METHOD DebounceOffHoldsOutputHighUntilElapsed
VAR
    fb : TcForge.FB_DigitalOutput;
END_VAR
TEST('DebounceOffHoldsOutputHighUntilElapsed');

// debounceOn stays at 0 so the output flushes HIGH immediately. The
// OFF-debounce (T#1S) then holds it HIGH even after SetOff, until TOF.Q
// falls — which it will not inside this synchronous test.
fb.cfg.debounceOff := T#1S;
fb.SetOn(eRequester := TcForge.E_Requester.PROG);
fb(inpQuality := TcForge.E_IO_Quality.GOOD);

AssertTrue(
    Condition := fb.sts.value,
    Message   := 'Precondition: SetOn with zero ON-debounce must flush HIGH');

fb.SetOff(eRequester := TcForge.E_Requester.PROG);
fb(inpQuality := TcForge.E_IO_Quality.GOOD);

AssertFalse(
    Condition := fb.sts.commanded,
    Message   := 'commanded must follow the SetOff request regardless of debounce');
AssertTrue(
    Condition := fb.sts.value,
    Message   := 'debounceOff must hold the physical output HIGH until the TOF expires');

TEST_FINISHED();
END_METHOD

METHOD InvertFlipsOutputInRegularMode
VAR
    fb : TcForge.FB_DigitalOutput;
END_VAR
TEST('InvertFlipsOutputInRegularMode');

// Active-low actuator: invert means "commanded ON -> physical LOW".
fb.cfg.invert := TRUE;
fb.SetOn(eRequester := TcForge.E_Requester.PROG);
fb(inpQuality := TcForge.E_IO_Quality.GOOD);

AssertTrue(
    Condition := fb.sts.commanded,
    Message   := 'commanded must reflect logical intent, not inverted physical output');
AssertFalse(
    Condition := fb.sts.value,
    Message   := 'invert must flip HIGH intent into a LOW physical output');

fb.SetOff(eRequester := TcForge.E_Requester.PROG);
fb(inpQuality := TcForge.E_IO_Quality.GOOD);

AssertFalse(
    Condition := fb.sts.commanded,
    Message   := 'commanded must follow SetOff regardless of invert');
AssertTrue(
    Condition := fb.sts.value,
    Message   := 'invert must flip LOW intent into a HIGH physical output');

TEST_FINISHED();
END_METHOD

METHOD BadQualityHoldsLastKnownGoodOutput
VAR
    fb : TcForge.FB_DigitalOutput;
END_VAR
TEST('BadQualityHoldsLastKnownGoodOutput');
fb.cfg.holdOnBadQuality := TRUE;

// Establish HIGH under GOOD quality.
fb.SetOn(eRequester := TcForge.E_Requester.PROG);
fb(inpQuality := TcForge.E_IO_Quality.GOOD);
AssertTrue(
    Condition := fb.sts.value,
    Message   := 'Precondition: SetOn under GOOD quality must drive HIGH');

// Now drop to BAD and try to SetOff. The hardware write must be skipped
// so the actuator stays in its last-known-good state.
fb.SetOff(eRequester := TcForge.E_Requester.PROG);
fb(inpQuality := TcForge.E_IO_Quality.BAD);

AssertTrue(
    Condition := fb.sts.value,
    Message   := 'BAD quality must hold the last-known-good physical output (no hardware write)');
AssertEquals_USINT(
    Expected := TcForge.E_IO_Quality.BAD,
    Actual   := fb.sts.quality,
    Message  := 'quality must surface the BAD tag to downstream consumers');

TEST_FINISHED();
END_METHOD

METHOD StsCommandedMirrorsRequestEvenUnderBadQuality
VAR
    fb : TcForge.FB_DigitalOutput;
END_VAR
TEST('StsCommandedMirrorsRequestEvenUnderBadQuality');
fb.cfg.holdOnBadQuality := TRUE;

// Even when the hardware write is vetoed by quality, commanded must
// still echo the live request so HMIs can show "operator asked for OFF
// but the output is held HIGH because quality is BAD".
fb.SetOn(eRequester := TcForge.E_Requester.PROG);
fb(inpQuality := TcForge.E_IO_Quality.GOOD);
fb.SetOff(eRequester := TcForge.E_Requester.PROG);
fb(inpQuality := TcForge.E_IO_Quality.BAD);

AssertFalse(
    Condition := fb.sts.commanded,
    Message   := 'commanded must reflect the current request even when BAD quality blocks the hardware write');
AssertTrue(
    Condition := fb.sts.value,
    Message   := 'value must still show the held physical output');

TEST_FINISHED();
END_METHOD

METHOD EdgePulsesAreOneScanWide
VAR
    fb : TcForge.FB_DigitalOutput;
END_VAR
TEST('EdgePulsesAreOneScanWide');

// Rising-edge pulse appears the cycle the physical output goes HIGH and
// is gone the next cycle.
fb.SetOn(eRequester := TcForge.E_Requester.PROG);
fb(inpQuality := TcForge.E_IO_Quality.GOOD);
AssertTrue(
    Condition := fb.sts.risingEdge,
    Message   := 'risingEdge must fire on the cycle the physical output goes HIGH');
AssertFalse(
    Condition := fb.sts.fallingEdge,
    Message   := 'fallingEdge must stay LOW on a rising edge cycle');

fb(inpQuality := TcForge.E_IO_Quality.GOOD);
AssertFalse(
    Condition := fb.sts.risingEdge,
    Message   := 'risingEdge must be exactly one scan wide');

// Falling edge on the way back down.
fb.SetOff(eRequester := TcForge.E_Requester.PROG);
fb(inpQuality := TcForge.E_IO_Quality.GOOD);
AssertTrue(
    Condition := fb.sts.fallingEdge,
    Message   := 'fallingEdge must fire on the cycle the physical output goes LOW');

fb(inpQuality := TcForge.E_IO_Quality.GOOD);
AssertFalse(
    Condition := fb.sts.fallingEdge,
    Message   := 'fallingEdge must be exactly one scan wide');

TEST_FINISHED();
END_METHOD

METHOD SinglePulseFiresOnCommandAndCanBeCanceled
VAR
    fb : TcForge.FB_DigitalOutput;
END_VAR
TEST('SinglePulseFiresOnCommandAndCanBeCanceled');

// SinglePulse with a long pulse width (T#10S) so the _tonPulseOn.Q
// stays FALSE inside this synchronous test and we observe the pulse
// while it is active.
fb.cfg.mode    := TcForge.E_DigitalOutput_Mode.SinglePulse;
fb.cfg.pulseOn := T#10S;

fb.SetOn(eRequester := TcForge.E_Requester.PROG);
fb(inpQuality := TcForge.E_IO_Quality.GOOD);

AssertTrue(
    Condition := fb.sts.value,
    Message   := 'SinglePulse must arm on the commanded rising edge and drive HIGH while active');

